                	ELSIF info.ClampA_Setting.PlaceArea = E_FeedInEmptyBox_PlaceArea.SameSizeConveyor THEN
                    	IF Input.bSameSizeCV_BoxNearStorageSensor THEN
                        	SlideClear_1st := FALSE;
                    	ELSE
                        	SlideClear_1st := TRUE;
                    	END_IF
                	END_IF
					IF SlideClear_1st  THEN
                		uiPlaceBothStep := 40;
					END_IF
//				ELSE
//					SlideClear_1st := FALSE;
//				END_IF
				IF Robot._DI1.Error THEN
					uiResumeStep := 81000;	// 補 missing assignment:雷射觸發 Robot.Error 走這條 abort 路徑時,uiResumeStep 必須設成本 step,否則 ABORTING/ABORTED 會用前一階段(pickup)的舊值,resume 跳回 pickup → 撞機
					uiResumePlaceBothStep := 0;
					SlideClear_1st		  := FALSE;
					_Abort	  := TRUE;
					strStatus := CONCAT('FB_FeedInEmptyBoxWithRobot_V3 Step 81000:',Robot.ErrMsg);
				END_IF
            40: //setup for clampB				
			
				CASE Info.ClampB_Setting.PlaceArea OF
					E_FeedInEmptyBox_PlaceArea.DiffSizeConveyor:
						WorkingConveyor REF= DiffSizeCV;
					E_FeedInEmptyBox_PlaceArea.SameSizeConveyor:
						WorkingConveyor REF= SameSizeCV;
				END_CASE
				IF __ISVALIDREF(WorkingConveyor) THEN
					uiPlaceBothStep := 50;
				END_IF
				IF Robot._DI1.Error THEN
					uiResumeStep := 81000;	// 補 missing assignment:雷射觸發 Robot.Error 走這條 abort 路徑時,uiResumeStep 必須設成本 step,否則 ABORTING/ABORTED 會用前一階段(pickup)的舊值,resume 跳回 pickup → 撞機
					uiResumePlaceBothStep := 0;
					SlideClear_1st		  := FALSE;
					_Abort	  := TRUE;
					strStatus := CONCAT('FB_FeedInEmptyBoxWithRobot_V3 Step 81000:',Robot.ErrMsg);
				END_IF

			50://Wait Robot finish clampA
				IF Robot._DI1.Notification THEN
					uiPlaceBothStep:=60;
				END_IF
				IF Robot._DI1.Error THEN
					uiResumeStep := 81000;	// 補 missing assignment:雷射觸發 Robot.Error 走這條 abort 路徑時,uiResumeStep 必須設成本 step,否則 ABORTING/ABORTED 會用前一階段(pickup)的舊值,resume 跳回 pickup → 撞機
					uiResumePlaceBothStep := 0;
					SlideClear_1st		  := FALSE;
					_Abort	  := TRUE;
					strStatus := CONCAT('FB_FeedInEmptyBoxWithRobot_V3 Step 81000:',Robot.ErrMsg);
				END_IF

			60://Move conveyor forward
				bWorkingConveyorMoveForward:=  TRUE;
				IF WorkingConveyor.InForWard THEN
					uiPlaceBothStep:=70;
				END_IF
				
			70://Update sensor
				M_UpdateConveyorSensor(Info.ClampB_Setting.PlaceArea);
				tonPlaceSensorDelay.IN := NOT SelectedSensor AND WorkingConveyor.InForWard ;
				IF 	tonPlaceSensorDelay.Q THEN
					tonPlaceSensorDelay.IN:=FALSE;
					uiPlaceBothStep:=80;
				END_IF
				
			80://Stop conveyor
				WorkingConveyor.M_MotorStop(); 
				bWorkingConveyorMoveForward:= FALSE;
				bWorkingConveyorMoveBackward :=FALSE; 
//				IF WorkingConveyor.InStopped THEN
//					uiPlaceBothStep:=90;
//				END_IF
				uiPlaceBothStep:=90;
			90:		
				WorkingConveyor.M_MotorStop(); 
				bWorkingConveyorMoveForward:= FALSE;
				bWorkingConveyorMoveBackward :=FALSE; 
//				IF	WorkingConveyor.InStopped THEN
               		 IF info.ClampB_Setting.PlaceArea = E_FeedInEmptyBox_PlaceArea.DiffSizeConveyor THEN
                 	   IF Input.bDifferentSizeCV_BoxDetect7_Sensor THEN						
                    	    SlideClear_2nd := FALSE;
                   		 ELSE                        
							SlideClear_2nd := TRUE;							
                   		 END_IF
					
               		 ELSIF info.ClampB_Setting.PlaceArea = E_FeedInEmptyBox_PlaceArea.SameSizeConveyor THEN
                 	   IF Input.bSameSizeCV_BoxNearStorageSensor THEN
                 	       SlideClear_2nd := FALSE;
                 		ELSE
							SlideClear_2nd := TRUE;
							
                  		END_IF
               			 END_IF
//				END_IF
				
				IF SlideClear_2nd THEN
                	uiPlaceBothStep := 99;
					tonPlaceSensorDelay.IN :=FALSE;
				END_IF
				IF Robot._DI1.Error THEN
						uiResumeStep := 81000;	// 補 missing assignment:雷射觸發 Robot.Error 走這條 abort 路徑時,uiResumeStep 必須設成本 step,否則 ABORTING/ABORTED 會用前一階段(pickup)的舊值,resume 跳回 pickup → 撞機
						uiResumePlaceBothStep := 60;
						SlideClear_2nd		  := FALSE;
						_Abort	  := TRUE;
						strStatus := CONCAT('FB_FeedInEmptyBoxWithRobot_V3 Step 81000:',Robot.ErrMsg);
					END_IF

			99:
				IF Robot._DI1.Error THEN
					uiResumeStep := 81000;	// 補 missing assignment:雷射觸發 Robot.Error 走這條 abort 路徑時,uiResumeStep 必須設成本 step,否則 ABORTING/ABORTED 會用前一階段(pickup)的舊值,resume 跳回 pickup → 撞機
					uiResumePlaceBothStep := 60;
					SlideClear_2nd		  := FALSE;
					_Abort	  := TRUE;
					strStatus := CONCAT('FB_FeedInEmptyBoxWithRobot_V3 Step 81000:',Robot.ErrMsg);
				END_IF
        // wait reset
        END_CASE
		bTimeOutIN :=TRUE;	
        IF NOT Robot._DI1.Done THEN
            Robot.M_StartMoveBoxToFeedInConveyor_ClampBoth(ClampA_Address := info.ClampA_Setting.PlaceArea,
                                                           ClampB_Address := info.ClampB_Setting.PlaceArea,
                                                           SlideClear_1st := SlideClear_1st,
                                                           SlideClear_2nd := SlideClear_2nd);
        ELSE
			bTimeOutIN:=FALSE;
            uiExecutingStep := 90000;
        END_IF
			
		IF tonTimeOut.Q THEN
			bTimeOutIN:=FALSE;
			_Abort :=TRUE;	
			uiResumeStep:=81000;		
			strStatus :='FB_FeedInEmptyBoxWithRobot_V3 Step 81000: Place Box timeout';
		END_IF
		IF Robot._DI1.Error THEN
			bTimeOutIN  := FALSE;
			_Abort 		:= TRUE;
			uiResumeStep:= 81000;
			strStatus	:= concat('FB_FeedInEmptyBoxWithRobot_V3 Step 81000:',Robot.ErrMsg);
			//strStatus	:= 'Test ErrMsg';
		END_IF
	
	90000: // Move conveyor forward a bit
		bWorkingConveyorMoveForward:=TRUE;
		IF WorkingConveyor.InForWard THEN
			uiExecutingStep := 91000;
		END_IF
	
	91000:// DELAY
		tonPlaceSensorDelay.PT:=T#0.8S;
		tonPlaceSensorDelay.IN :=TRUE;
		IF tonPlaceSensorDelay.Q THEN
			uiExecutingStep := 92000;
		END_IF
	
	92000:// STOP MOTOR
		tonPlaceSensorDelay.IN :=FALSE;
		bWorkingConveyorMoveForward:=FALSE;
		WorkingConveyor.M_MotorStop();
		IF WorkingConveyor.InStopped THEN
			uiExecutingStep := 99000;
		END_IF
			
				
    99000: // process done
        // Stop FeedIn conveyor
		tonFeedInConveyorDelay.IN :=TRUE;		//Delay FeedInConveyor stop 500MS Edit by Min
		IF tonFeedInConveyorDelay.Q THEN
			DAS_CoreSys.MachineControl.fballocatearea.M_ReleasePulloutAccess(ControlAccess := E_RoundBeltControlAccess.FanucRobot);
			DiffSizeCV.M_MotorStop();
			SameSizeCV.M_MotorStop();
			bWorkingConveyorMoveForward:=FALSE;
			tonFeedInConveyorDelay.IN :=FALSE;
			Status    := 'FB_FeedInEmptyBoxWithRobot_V3 Step 99000: Process completed';
				IF DiffSizeCV.InStopped AND SameSizeCV.InStopped THEN
				 _Executed := TRUE;
				END_IF
		END_IF
END_CASE

// 移植 mirror V4 (commit 326aa68): _Executed 判斷加 NOT Robot.Halt 防止暫停期間誤跳 DONE;
// 新增 ELSIF Pause 進 STATE_Holding,啟動 PackML 暫停流程
IF _Executed AND NOT Robot.Halt THEN
    eState := STATE_DONE;
ELSIF NOT Execute THEN
    eState := STATE_RESETTING;
ELSIF Pause THEN
	bPauseLatched := TRUE;
	uiPauseFromStep := uiExecutingStep;
	_HoldingCompleted := FALSE;
	_HeldCompleted := FALSE;
	_UnholdCompleted := FALSE;
	uiHoldingStep := 0;
	uiHeldStep := 0;
	uiUnholdStep := 0;
	eState := STATE_Holding;
ELSIF Abort OR _Abort THEN
	//FUN_UniqueErrorCodeGenerator(iErrorID := ErrorID,UinqueErrorCode=>_UniqueErrorCode);
	eState := STATE_ABORTING;
ELSIF _Error THEN
	//FUN_UniqueErrorCodeGenerator(iErrorID := ErrorID,UinqueErrorCode=>_UniqueErrorCode);
	eState := STATE_ERROR;
END_IF
END_METHOD

METHOD M_STATE_HELD
VAR_INPUT
END_VAR
Busy := FALSE;
Paused := TRUE;
Status := 'Paused';

IF NOT Execute THEN
	eState := STATE_RESETTING;
ELSIF Abort OR _Abort THEN
	eState := STATE_ABORTING;
ELSIF _Error THEN
	eState := STATE_ERROR;
ELSIF NOT Pause THEN
	_UnholdCompleted := FALSE;
	uiUnholdStep := 0;
	eState := STATE_UnHold;
END_IF
END_METHOD

METHOD M_STATE_HOLDING
VAR_INPUT
END_VAR
Busy := TRUE;
Paused := FALSE;
Status := 'Pause holding';

bTimeOutIN := FALSE;
tonPlaceSensorDelay.IN := FALSE;
tonFeedInConveyorDelay.IN := FALSE;
bWorkingConveyorMoveForward := FALSE;
bWorkingConveyorMoveBackward := FALSE;

CASE uiHoldingStep OF
	0:
		CASE uiExecutingStep OF
			0,10,20,1000,1100:
				uiHoldingStep := 9999;

			61000,71000,81000,90000,91000,92000:
				IF __ISVALIDREF(WorkingConveyor) THEN
					WorkingConveyor.M_MotorStop();
					IF WorkingConveyor.InStopped THEN
						uiHoldingStep := 9999;
					END_IF
				ELSE
					DiffSizeCV.M_MotorStop();
					SameSizeCV.M_MotorStop();
					IF DiffSizeCV.InStopped AND SameSizeCV.InStopped THEN
						uiHoldingStep := 9999;
					END_IF
				END_IF

			99000:
				DAS_CoreSys.MachineControl.fballocatearea.M_ReleasePulloutAccess(
					ControlAccess := E_RoundBeltControlAccess.FanucRobot);
				DiffSizeCV.M_MotorStop();
				SameSizeCV.M_MotorStop();
				IF DiffSizeCV.InStopped AND SameSizeCV.InStopped THEN
					_Executed := TRUE;
					uiHoldingStep := 9999;
				END_IF

		ELSE
			DAS_CoreSys.MachineControl.fballocatearea.M_StopStoragePulloutAction();
			IF Robot.Halt OR Robot._DI1.Done OR NOT Robot._DI12.BzoneInWork THEN
				uiHoldingStep := 9999;
			END_IF
		END_CASE

	9999:
		_HoldingCompleted := TRUE;
END_CASE

IF NOT Execute THEN
	eState := STATE_RESETTING;
ELSIF Abort OR _Abort THEN
	eState := STATE_ABORTING;
ELSIF _Error THEN
	eState := STATE_ERROR;
ELSIF _Executed THEN
	eState := STATE_DONE;
ELSIF _HoldingCompleted THEN
	eState := STATE_Held;
END_IF
END_METHOD

METHOD  M_STATE_RESETTING
VAR_INPUT
END_VAR
IF _Executed THEN Done :=TRUE ; END_IF
CASE uiResettingStep OF
	0:
		//DAS.fbStorageArea.M_InactivePulloutConveyorInternCtrl();
		Robot.M_ResetAllCommand();
		Robot.Bzone_AllowWork:=FALSE;
		DiffSizeCV.M_MotorStop();
		SameSizeCV.M_MotorStop();
		 DAS_CoreSys.MachineControl.fballocatearea.M_ReleasePulloutAccess(ControlAccess := E_RoundBeltControlAccess.FanucRobot);
		 DAS_CoreSys.MachineControl.fballocatearea.M_StopStoragePulloutAction();
		WareHouse.M_ResetFeedInBox();
		WareHouse.M_ResetReloadBox();
		bWorkingConveyorMoveForward  :=FALSE;
		bWorkingConveyorMoveBackward :=FALSE;
		bTimeOutIN:=FALSE;
		Paused := FALSE;
		bPauseLatched := FALSE;
		uiPauseFromStep := 0;
		AClampMoveDone	:= FALSE;
		BClampMoveDone	:= FALSE;
		_AClampDoingWork	:= FALSE;
		_BClampDoingWork	:= FALSE;
		uiResettingStep := 100;
	100:
		_ResetCompleted := TRUE;
END_CASE
IF _ResetCompleted THEN
    eState := STATE_DORMANT;
END_IF
END_METHOD

METHOD M_STATE_UNHOLD
VAR_INPUT
END_VAR
Paused := FALSE;
Status := '';
tonPlaceSensorDelay.IN := FALSE;
tonFeedInConveyorDelay.IN := FALSE;
_UnholdCompleted := TRUE;

IF _UnholdCompleted THEN
	eState := STATE_EXECUTING;
END_IF
END_METHOD

METHOD PRIVATE M_UpdateConveyorSensor : BOOL
VAR_INPUT
	Area : E_FeedInEmptyBox_PlaceArea;
END_VAR
CASE Area OF
	
	E_FeedInEmptyBox_PlaceArea.SameSizeConveyor :
		SelectedSensor := Input.bSameSizeCV_BoxNearStorageSensor ;
	
	E_FeedInEmptyBox_PlaceArea.DiffSizeConveyor:
		SelectedSensor := Input.bDifferentSizeCV_BoxDetect7_Sensor;
END_CASE
END_METHOD

END_FUNCTION_BLOCK

// ---- Library/20_MachineUnits/21_StorageArea/Service_Robot/FB_ReloadRoundBeltBoxWithRobot_V2.TcPOU
FUNCTION_BLOCK FB_ReloadRoundBeltBoxWithRobot_V2 EXTENDS FB_ObjectBase_V2 IMPLEMENTS IBasicElement
VAR_INPUT
    // Below are the components being controlled.
    Robot         : REFERENCE TO FB_FanucRobot_Basic_V2; // Fanuc Robot
    //AllocatedArea : REFERENCE TO FB_AllocatingSpace; // Allocated area , use to control round belt
	RoundBelt	: REFERENCE TO FB_RoundBeltService;
    WareHouse     : REFERENCE TO FB_WareHouse; // Storage area warehouse A and warehouse B conveyor and sensor
    //	A2_Sensor : REFERENCE TO FB_Sensor;
    //	A3_Sensor : REFERENCE TO FB_Sensor;
	Input : ST_InputTable;
    Info : ST_ReloadRoundBeltBox_Info; // Setting the feedin emptybox action's parameter
    Stop : BOOL;
END_VAR
VAR_OUTPUT
	AClampMoveDone	: BOOL;
	BClampMoveDone	: BOOL;
END_VAR
VAR
    strStatus         : STRING;
    tonTimeOut        : TON;
    tonFeedBoxTimeout : TON;
    _UniqueErrorCode  : STRING;
    PreviousStrStatus : STRING;
    PreviousErrorCode : STRING;
    A2_Sensor         : BOOL;
    A3_Sensor         : BOOL;
	//_Abort			  : BOOL;

	// Clamp work
	_AClampDoingWork	: BOOL;
	_BClampDoingWork	: BOOL;

	// ========== Resume 續做機制 ==========
	uiResumeStep	: UDINT := 0;	// 錯誤發生時記錄的步驟，供續做使用
	
	_bRetry			: BOOL;
END_VAR

SUPER^.A10_StateControl();
A00_BasicUnits();
A2_Sensor := Input.bRoundBelt_ChangeZoneA2Detect_Sensor;
A3_Sensor := Input.bRoundBelt_ChangeZoneA3Detect_Sensor;

(*============================================================
Create Date : 2025/11/22
Last Update	: 2026/03/31
Change Log  : 2025/11/24，send flag A clamp done and B clamp done for C# use to SQL // Owner : Gamin
			  2026/03/31，移植泰興鏡射版本，雷射續做，清除手臂錯誤。
============================================================*)

ACTION A00_BasicUnits:
tonTimeOut(PT:=T#60S);
tonFeedBoxTimeout(PT:=T#15s);
END_ACTION

METHOD M_CheckCommand : BOOL
VAR_INPUT
END_VAR
VAR_INST
	CheckBehavior : BOOL; // True :Behavior is correct
END_VAR
VAR
	I: INT;
END_VAR
// Memory clear
CheckBehavior := FALSE;
// Check command is correct
IF info.ClampA_Setting.Behavior = E_ClampWork.Work OR info.ClampB_Setting.Behavior = E_ClampWork.Work THEN
	CheckBehavior := TRUE;
ELSE
	CheckBehavior := FALSE;
END_IF


M_CheckCommand := CheckBehavior;
END_METHOD

METHOD M_CheckUnitsNotBusy : BOOL
VAR_INPUT
END_VAR
M_CheckUnitsNotBusy := true;
END_METHOD

METHOD M_CheckUnitsReady : BOOL
VAR_INPUT
END_VAR
M_CheckUnitsReady := true;
END_METHOD

METHOD M_SelectActionMode : E_ReloadRoundBoxAction
VAR_INPUT
END_VAR
IF info.ClampA_Setting.Behavior <> E_ClampWork.Work AND info.ClampB_Setting.Behavior <> E_ClampWork.Work THEN
	M_SelectActionMode :=E_ReloadRoundBoxAction.Undefined;
ELSIF info.ClampA_Setting.Behavior = E_ClampWork.Work AND info.ClampB_Setting.Behavior <> E_ClampWork.Work THEN
	IF info.ClampA_Setting.PickUpArea = E_ReloadRoundBelt_PickupArea.WareHouseA THEN
		M_SelectActionMode := E_ReloadRoundBoxAction.ClampA_WareHouseA;
	ELSIF info.ClampA_Setting.PickUpArea = E_ReloadRoundBelt_PickupArea.WareHouseB THEN
		M_SelectActionMode := E_ReloadRoundBoxAction.ClampA_WareHouseB;
	END_IF
ELSIF info.ClampA_Setting.Behavior <> E_ClampWork.Work AND info.ClampB_Setting.Behavior = E_ClampWork.Work THEN
	IF info.ClampB_Setting.PickUpArea = E_ReloadRoundBelt_PickupArea.WareHouseA THEN
		M_SelectActionMode := E_ReloadRoundBoxAction.ClampB_WareHouseA;
	ELSIF info.ClampB_Setting.PickUpArea = E_ReloadRoundBelt_PickupArea.WareHouseB THEN
		M_SelectActionMode := E_ReloadRoundBoxAction.ClampB_WareHouseB;
	END_IF
ELSIF info.ClampA_Setting.Behavior = E_ClampWork.Work AND info.ClampB_Setting.Behavior = E_ClampWork.Work THEN
	IF info.ClampA_Setting.PickUpArea = E_ReloadRoundBelt_PickupArea.WareHouseA THEN
		IF info.ClampB_Setting.PickUpArea = E_ReloadRoundBelt_PickupArea.WareHouseA THEN
			M_SelectActionMode := E_ReloadRoundBoxAction.A_WareHouseA_B_WareHouseA;
		ELSIF info.ClampB_Setting.PickUpArea = E_ReloadRoundBelt_PickupArea.WareHouseB THEN
			M_SelectActionMode := E_ReloadRoundBoxAction.A_WareHouseA_B_WareHouseB;
		END_IF
	ELSIF info.ClampA_Setting.PickUpArea = E_ReloadRoundBelt_PickupArea.WareHouseB THEN
		IF info.ClampB_Setting.PickUpArea = E_ReloadRoundBelt_PickupArea.WareHouseA THEN
			M_SelectActionMode := E_ReloadRoundBoxAction.A_WareHouseB_B_WareHouseA;
		ELSIF info.ClampB_Setting.PickUpArea = E_ReloadRoundBelt_PickupArea.WareHouseB THEN
			M_SelectActionMode := E_ReloadRoundBoxAction.A_WareHouseB_B_WareHouseB;
		END_IF
	END_IF
END_IF
END_METHOD

METHOD  M_STATE_ABORTED
VAR_INPUT
END_VAR
IF NOT _bRetry THEN
	Busy    := FALSE;
	Error	:= TRUE;
	Aborted := TRUE;
	_Abort  := TRUE;
	UniqueErrorCode := _UniqueErrorCode;
	Status := strStatus;
	_AbortCompleted := FALSE;
	uiAbortingStep	:= 0;
END_IF

IF Reset THEN
	_bRetry := TRUE;
	Error	:= FALSE;
	Aborted := FALSE;
	_Abort  := FALSE;
END_IF

// ============================================================
// Resume 機制：保持 Execute 並按 Reset 可從錯誤點繼續
// ============================================================
IF NOT Execute THEN
	eState := STATE_RESETTING;
ELSIF Execute AND _bRetry AND NOT Robot._DI1.Error AND NOT Robot.Halt THEN
	// Resume 模式：確認 Robot 不在暫停且無錯誤，從儲存的步驟繼續執行
	Status := '';

	uiExecutingStep := uiResumeStep;
	PreviousStrStatus := strStatus;
	PreviousErrorCode := _UniqueErrorCode;
	
	IF GVL_ADS.MachineState <>E_MachineState.Error THEN
		eSTATE:=STATE_EXECUTING;
	END_IF
END_IF
END_METHOD

METHOD  M_STATE_ABORTING
VAR_INPUT
END_VAR
CASE uiAbortingStep OF
	0:
			_Abort  := FALSE;
			_bRetry := FALSE;
			tonTimeOut.IN 		 := FALSE;
			tonFeedBoxTimeout.IN := FALSE;

			uiAbortingStep := 100;
	
    100:
			IF Robot._DI1.Error THEN
				uiAbortingStep := 200;
			ELSE
				uiAbortingStep := 9999;
			END_IF
	200:		
			 IF DAS_CoreSys.MachineControl.M_RobotResetCmd() THEN
				 uiAbortingStep := 300;
			 END_IF
	300:
			IF DAS_CoreSys.MachineControl.M_RobotStartCmd() THEN
				 uiAbortingStep := 400;
			 END_IF 
	400:
			IF Robot._DI1.Error THEN
		 		uiAbortingStep := 200;
			ELSE
				uiAbortingStep := 9999;
			END_IF
	9999:
			_AbortCompleted := TRUE;
END_CASE


IF _AbortCompleted THEN
    eState := STATE_Aborted;
END_IF
END_METHOD

METHOD  M_STATE_DONE
VAR_INPUT
END_VAR
Busy   := FALSE;
_Error := Error := FALSE;
_Abort := Abort := FALSE;
Done   := TRUE;

IF NOT Execute THEN
    eState := STATE_RESETTING;
END_IF
END_METHOD

METHOD  M_STATE_DORMANT
VAR_INPUT
END_VAR
// Clear FB output
Busy            := FALSE;
Done            := FALSE;
Aborted         := FALSE;
Error           := FALSE;
ErrorID         := 0;
Status          := '';
_ResetCompleted := FALSE;
_Error          := FALSE;
_Executed       := FALSE;
_Abort			:= FALSE;
uiExecutingStep := 0;
uiResettingStep := 0;
uiResumeStep    := 0;	// 清除 Resume 步驟
uiAbortingStep	:= 0;
tonTimeOut.IN := FALSE;
tonFeedBoxTimeout.IN := FALSE;
PreviousStrStatus := '';
PreviousErrorCode := '';
_UniqueErrorCode := '0';
AClampMoveDone := FALSE;
BClampMoveDone := FALSE;
_AClampDoingWork := FALSE;
_BClampDoingWork := FALSE;
_AbortCompleted	 := FALSE;
_bRetry			 := FALSE;

// Wait Execute command
IF Execute AND NOT stop THEN
    eState := STATE_EXECUTING;
END_IF
END_METHOD

METHOD  M_STATE_ERROR
VAR_INPUT
END_VAR
UniqueErrorCode	:= _UniqueErrorCode;
Error			:= TRUE;
status			:= strStatus;
Busy			:= FALSE;

IF NOT Execute THEN
    eState := STATE_RESETTING;
END_IF
END_METHOD

METHOD M_STATE_EXECUTING
VAR_INPUT
END_VAR
VAR_INST
    ActionMode       : E_ReloadRoundBoxAction;
	BoxReady_1st : BOOL;
	BoxReady_2nd : BOOL;
    CarrierReady_1st : BOOL;
    CarrierReady_2nd : BOOL;
    uiPickUpBothStep : UINT;
    uiPlaceBothStep  : UINT;
    ClampA_WareHouseCoordinates : ST_WareHouseCoordinates;
    ClampB_WareHouseCoordinates : ST_WareHouseCoordinates;
	
	//=============== test only====
		_A2Sensor	:BOOL;
		_A3Sensor	:BOOL;
END_VAR
// Set status busy
Busy := TRUE;
IF THIS^.Stop THEN // Pending the timeout when Stop signal occur
	tonTimeout.IN :=FALSE;
END_IF
CASE uiExecutingStep OF
    0:
        // Clear variable
        ActionMode       := E_ReloadRoundBoxAction.Undefined;
        CarrierReady_1st := FALSE;
        CarrierReady_2nd := FALSE;
        uiPickUpBothStep := 0;
        uiPlaceBothStep  := 0;
		BoxReady_1st := 0;
		BoxReady_2nd := 0;
        // Check command
        IF M_CheckCommand() THEN
            uiExecutingStep := 10;
        END_IF
    10:
        // Start process, check units first
        IF M_CheckUnitsReady() THEN
            uiExecutingStep := 20;
        END_IF
    20:
        // CHeck units not busy state
        IF M_CheckUnitsNotBusy() THEN
            uiExecutingStep := 1000;
        END_IF
    1000:
        // Select action mode
        ActionMode      := M_SelectActionMode();
        uiExecutingStep := 1100;
    1100:
		//DAS_CoreSys.MachineControl.fbAllocateArea.M_ActiveRoundBeltInternalCtrl(); //Request round belt 
		DAS_CoreSys.MachineControl.fbAllocateArea.M_GetRoundBeltAccess(ControlAccess := E_RoundBeltControlAccess.FanucRobot);
        CASE ActionMode OF
            E_ReloadRoundBoxAction.ClampA_WareHouseA:
                uiExecutingStep := 10000;
            E_ReloadRoundBoxAction.ClampA_WareHouseB:
                uiExecutingStep := 11000;
            E_ReloadRoundBoxAction.ClampB_WareHouseA:
                uiExecutingStep := 20000;
            E_ReloadRoundBoxAction.ClampB_WareHouseB:
                uiExecutingStep := 21000;
            E_ReloadRoundBoxAction.A_WareHouseA_B_WareHouseA:
                uiExecutingStep := 30000;
            E_ReloadRoundBoxAction.A_WareHouseA_B_WareHouseB:
                uiExecutingStep := 31000;
            E_ReloadRoundBoxAction.A_WareHouseB_B_WareHouseA:
                uiExecutingStep := 32000;
            E_ReloadRoundBoxAction.A_WareHouseB_B_WareHouseB:
                uiExecutingStep := 33000;
        END_CASE
    10000: // Only ClampA pickup box from WarehouseA
        IF NOT Robot._DI1.Done THEN
            // Read ClampA Warehouse coordinate
            ClampA_WareHouseCoordinates := info.ClampA_Setting.WareHouseSetting;
            // Reload Warehouse target position box
            WareHouse.M_StartReloadBox(WareHouseSelect := E_WareHouse.WareHouseA, WarehouseCoordinates := ClampA_WareHouseCoordinates);

            // Check Box reload completed
            IF WareHouse.bReloadBox_Completed THEN
                BoxReady_1st 	 := TRUE;
				_AClampDoingWork := TRUE;
            END_IF

            // Robot Warehouse move
            Robot.M_StartWareHousePickUpBox_ClampA(WareHouseSelect := E_WareHouse.WareHouseA,
                                                   Info            := ClampA_WareHouseCoordinates,
                                                   BoxReady_1st    := BoxReady_1st);

            DAS_CoreSys.MachineControl.fbAllocateArea.M_GetRoundBeltAccess(ControlAccess := E_RoundBeltControlAccess.FanucRobot);
            DAS_CoreSys.MachineControl.fbAllocateArea.M_StartReloadRoundBeltAtion(ReloadStation := info.ClampA_Setting.RoundBeltSetting.Station);
			
			// make sure robot doing AClamp done
			IF _AClampDoingWork AND  NOT Robot._DI1.ClampA_Open THEN
				AClampMoveDone := TRUE;
			END_IF
        ELSE
			tonTimeOut.IN :=FALSE;
            uiExecutingStep := 10080;
        END_IF
		tonTimeOut.IN :=TRUE;
		IF tonTimeOut.Q THEN
			uiResumeStep := 10000;
			_Abort := TRUE;
			tonTimeOut.IN :=FALSE;
			strStatus :='FB_ReloadRoundBeltBoxWithRobot_V2 Step 10000: Pick Box timeout';
		END_IF
    10080:
        Robot.M_ResetAllCommand(); // Clear command and go to place box
		WareHouse.M_ResetReloadBox();
        IF NOT Robot._DI1.Done THEN
            uiExecutingStep := 60000; // only place clampA
        END_IF
    11000: // Only ClampA pickup box from WarehouseB
        IF NOT Robot._DI1.Done THEN
            // Read ClampA Warehouse coordinate
            ClampA_WareHouseCoordinates := info.ClampA_Setting.WareHouseSetting;
            // Reload Warehouse target position box
            WareHouse.M_StartReloadBox(WareHouseSelect := E_WareHouse.WareHouseB, WarehouseCoordinates := ClampA_WareHouseCoordinates);

            // Check Box reload completed
            IF WareHouse.bReloadBox_Completed THEN
                BoxReady_1st 	 := TRUE;
				_AClampDoingWork := TRUE;
            END_IF

            // Robot Warehouse move
            Robot.M_StartWareHousePickUpBox_ClampA(WareHouseSelect := E_WareHouse.WareHouseB,
                                                   Info            := ClampA_WareHouseCoordinates,
                                                   BoxReady_1st    := BoxReady_1st);

            DAS_CoreSys.MachineControl.fbAllocateArea.M_GetRoundBeltAccess(ControlAccess := E_RoundBeltControlAccess.FanucRobot);
            DAS_CoreSys.MachineControl.fbAllocateArea.M_StartReloadRoundBeltAtion(ReloadStation := info.ClampA_Setting.RoundBeltSetting.Station);
			
			// make sure robot doing AClamp done
			IF _AClampDoingWork AND  NOT Robot._DI1.ClampA_Open THEN
				AClampMoveDone := TRUE;
			END_IF

        ELSE
			tonTimeOut.IN :=FALSE;
            uiExecutingStep := 11080;
        END_IF
		tonTimeOut.IN :=TRUE;
		IF tonTimeOut.Q THEN
			uiResumeStep := 11000;
			_Abort := TRUE;
			tonTimeOut.IN :=FALSE;
			strStatus :='FB_ReloadRoundBeltBoxWithRobot_V2 Step 11000: Pick Box timeout';
		END_IF
    11080:
        Robot.M_ResetAllCommand(); // Clear command and go to place box

        IF NOT Robot._DI1.Done THEN
            uiExecutingStep := 60000; // only place clampA
        END_IF
    20000: // Only ClampB pickup from WarehouseA
        IF NOT Robot._DI1.Done THEN
            // Read ClampA Warehouse coordinate
            ClampB_WareHouseCoordinates := info.ClampB_Setting.WareHouseSetting;
            // Reload Warehouse target position box
            WareHouse.M_StartReloadBox(WareHouseSelect := E_WareHouse.WareHouseA, WarehouseCoordinates := ClampB_WareHouseCoordinates);

            // Check Box reload completed
            IF WareHouse.bReloadBox_Completed THEN
                BoxReady_2nd 	 := TRUE;
				_BClampDoingWork := TRUE;
            END_IF

            // Robot Warehouse move
            Robot.M_StartWareHousePickUpBox_ClampB(WareHouseSelect := E_WareHouse.WareHouseA,
                                                   Info            := ClampB_WareHouseCoordinates,
                                                   BoxReady_2nd    := BoxReady_2nd);

          	DAS_CoreSys.MachineControl.fbAllocateArea.M_GetRoundBeltAccess(ControlAccess := E_RoundBeltControlAccess.FanucRobot);
            DAS_CoreSys.MachineControl.fbAllocateArea.M_StartReloadRoundBeltAtion(ReloadStation := info.ClampB_Setting.RoundBeltSetting.Station);
			
			// robot doing BClamp done
			IF _BClampDoingWork AND NOT Robot._DI1.ClampB_Open THEN 
				BClampMoveDone := TRUE;
			END_IF

        ELSE
			tonTimeOut.IN :=FALSE;
            uiExecutingStep := 20080;
        END_IF
			tonTimeOut.IN :=TRUE;
		IF tonTimeOut.Q THEN
			uiResumeStep := 20000;
			_Abort := TRUE;
			tonTimeOut.IN :=FALSE;
			strStatus :='FB_ReloadRoundBeltBoxWithRobot_V2 Step 20000: Pick Box timeout';
		END_IF
    20080:
        WareHouse.M_ResetReloadBox();
        Robot.M_ResetAllCommand();

        IF NOT Robot._DI1.Done THEN
            uiExecutingStep := 70000; // Only ClampB place box
        END_IF
    21000: // Only ClampB pickup from WarehouseB
        IF NOT Robot._DI1.Done THEN
            // Read ClampA Warehouse coordinate
            ClampB_WareHouseCoordinates := info.ClampB_Setting.WareHouseSetting;
            // Reload Warehouse target position box
            WareHouse.M_StartReloadBox(WareHouseSelect := E_WareHouse.WareHouseB, WarehouseCoordinates := ClampB_WareHouseCoordinates);

            // Check Box reload completed
            IF WareHouse.bReloadBox_Completed THEN
                BoxReady_2nd 	 := TRUE;
				_BClampDoingWork := TRUE;
            END_IF

            // Robot Warehouse move
            Robot.M_StartWareHousePickUpBox_ClampB(WareHouseSelect := E_WareHouse.WareHouseB,
                                                   Info            := ClampB_WareHouseCoordinates,
                                                   BoxReady_2nd    := BoxReady_2nd);
            DAS_CoreSys.MachineControl.fbAllocateArea.M_GetRoundBeltAccess(ControlAccess := E_RoundBeltControlAccess.FanucRobot);
            DAS_CoreSys.MachineControl.fbAllocateArea.M_StartReloadRoundBeltAtion(ReloadStation := info.ClampA_Setting.RoundBeltSetting.Station);
			
			// robot doing BClamp done
			IF _BClampDoingWork AND NOT Robot._DI1.ClampB_Open THEN 
				BClampMoveDone := TRUE;
			END_IF

        ELSE
			tonTimeOut.IN :=FALSE;
            uiExecutingStep := 21080;
        END_IF
			tonTimeOut.IN :=TRUE;
		IF tonTimeOut.Q THEN
			uiResumeStep := 21000;
			_Abort := TRUE;
			tonTimeOut.IN :=FALSE;
			strStatus :='FB_ReloadRoundBeltBoxWithRobot_V2 Step 21000: Pick Box timeout';
		END_IF
    21080:
        WareHouse.M_ResetReloadBox();
        Robot.M_ResetAllCommand();

        IF NOT Robot._DI1.Done THEN
            uiExecutingStep := 70000; // Only ClampB place box
        END_IF
    30000: // ClampA and ClampB pickup box from WarehouseA
        ClampA_WareHouseCoordinates := info.ClampA_Setting.WareHouseSetting;
        ClampB_WareHouseCoordinates := info.ClampB_Setting.WareHouseSetting;

        CASE uiPickUpBothStep OF
            0: // ClampA target slide move the box to front side
                WareHouse.M_StartReloadBox(WareHouseSelect      := E_WareHouse.WareHouseA,
                                           WarehouseCoordinates := ClampA_WareHouseCoordinates);

              	DAS_CoreSys.MachineControl.fbAllocateArea.M_GetRoundBeltAccess(ControlAccess := E_RoundBeltControlAccess.FanucRobot);
                DAS_CoreSys.MachineControl.fbAllocateArea.M_StartReloadRoundBeltAtion(ReloadStation := info.ClampA_Setting.RoundBeltSetting.Station);

                IF WareHouse.bReloadBox_Completed THEN
                    BoxReady_1st     := TRUE;
					_AClampDoingWork := TRUE;
                    uiPickUpBothStep := 10;
                END_IF

            10: // wait Robot Allow continue
                IF Robot._DI1.Notification AND
                    NOT
                    WareHouse._stWarehouseList.ASide_Layers[ClampA_WareHouseCoordinates.Layer].stStatus.bSlides[ClampA_WareHouseCoordinates.Slide]
                    THEN
                    WareHouse.M_ResetReloadBox();

                    IF NOT WareHouse.bReloadBox_Completed THEN
                        uiPickUpBothStep := 20;
                    END_IF

                END_IF
            20: // ClampB target slide move the box to front slide
                WareHouse.M_StartReloadBox(WareHouseSelect := E_WareHouse.WareHouseA, WarehouseCoordinates := ClampB_WareHouseCoordinates);

                IF WareHouse.bReloadBox_Completed THEN
                    BoxReady_2nd     := TRUE;
					_BClampDoingWork := TRUE;
                    uiPickUpBothStep := 99;
                END_IF
            99:
        // wait reset
        END_CASE

        Robot.M_StartWareHousePickUpBox_ClampBoth(WareHouseSelect := E_WareHouse.WareHouseA,
                                                  ClampA_Info     := ClampA_WareHouseCoordinates,
                                                  ClampB_Info     := ClampB_WareHouseCoordinates,
                                                  BoxReady_1st    := BoxReady_1st,
                                                  BoxReady_2nd    := BoxReady_2nd);
												  
		// robot doing AClamp done
			IF _AClampDoingWork AND  NOT Robot._DI1.ClampA_Open THEN
				AClampMoveDone := TRUE;
			END_IF

		// robot doing BClamp done
			IF _BClampDoingWork AND NOT Robot._DI1.ClampB_Open THEN 
				BClampMoveDone := TRUE;
			END_IF										  

        IF Robot._DI1.Done THEN
			tonTimeOut.IN :=FALSE;
            uiExecutingStep := 30080;
        END_IF
			tonTimeOut.IN :=TRUE;
		IF tonTimeOut.Q THEN
			uiResumeStep := 30000;
			_Abort := TRUE;
			tonTimeOut.IN :=FALSE;
			strStatus :='FB_ReloadRoundBeltBoxWithRobot_V2 Step 30000: Pick Box timeout';
		END_IF
    30080: // Check robot command is clear
        WareHouse.M_ResetReloadBox();
        Robot.M_ResetAllCommand();

        IF NOT Robot._DI1.Done THEN
            uiExecutingStep := 80000; // go to place step
        END_IF
    31000: // ClampA pickup from Warehouse A, ClampB pickup from Warehouse B
        IF NOT Robot._DI1.Done THEN
            ClampA_WareHouseCoordinates := info.ClampA_Setting.WareHouseSetting;
            WareHouse.M_StartReloadBox(WareHouseSelect := E_WareHouse.WareHouseA, WarehouseCoordinates := ClampA_WareHouseCoordinates);

            IF WareHouse.bReloadBox_Completed THEN
                BoxReady_1st     := TRUE;
				_AClampDoingWork := TRUE;
            END_IF
			DAS_CoreSys.MachineControl.fbAllocateArea.M_ActiveRoundBeltInternalCtrl();
			DAS_CoreSys.MachineControl.fbAllocateArea.M_StartReloadRoundBeltAtion(ReloadStation := info.ClampA_Setting.RoundBeltSetting.Station);
            Robot.M_StartWareHousePickUpBox_ClampA(WareHouseSelect := E_WareHouse.WareHouseA,
                                                   Info            := ClampA_WareHouseCoordinates,
                                                   BoxReady_1st    := BoxReady_1st);
			
			// robot doing AClamp done
			IF _AClampDoingWork AND  NOT Robot._DI1.ClampA_Open THEN
				AClampMoveDone := TRUE;
			END_IF						   
												   
        ELSE
			tonTimeOut.IN :=FALSE;
            uiExecutingStep := 31080;
        END_IF
			tonTimeOut.IN :=TRUE;
		IF tonTimeOut.Q THEN
			uiResumeStep := 31000;
			_Abort := TRUE;
			tonTimeOut.IN :=FALSE;
			strStatus :='FB_ReloadRoundBeltBoxWithRobot_V2 Step 31000: Pick Box timeout';
		END_IF

    31080:
        Robot.M_ResetAllCommand(); // Clear command and go to place box
		WareHouse.M_ResetReloadBox();
        IF NOT Robot._di1.Done THEN
            uiExecutingStep := 31100; // ClampA pickup finished, ClampB pickup start
        END_IF
    31100:
        IF NOT Robot._di1.Done THEN
            ClampB_WareHouseCoordinates := info.ClampB_Setting.WareHouseSetting;
            WareHouse.M_StartReloadBox(WareHouseSelect := E_WareHouse.WareHouseB, WarehouseCoordinates := ClampB_WareHouseCoordinates);

            IF WareHouse.bReloadBox_Completed THEN
                BoxReady_2nd 	 := TRUE;
				_BClampDoingWork := TRUE;
            END_IF

            Robot.M_StartWareHousePickUpBox_ClampB(WareHouseSelect := E_WareHouse.WareHouseB,
                                                   Info            := ClampB_WareHouseCoordinates,
                                                   BoxReady_2nd    := BoxReady_2nd);
												   
			// robot doing BClamp done
			IF _BClampDoingWork AND NOT Robot._DI1.ClampB_Open THEN 
				BClampMoveDone := TRUE;
			END_IF
												   
        ELSE
			tonTimeOut.IN :=FALSE;
            uiExecutingStep := 31180;
        END_IF
				tonTimeOut.IN :=TRUE;
		IF tonTimeOut.Q THEN
			uiResumeStep := 31100;
			_Abort := TRUE;
			tonTimeOut.IN :=FALSE;
			strStatus :='FB_ReloadRoundBeltBoxWithRobot_V2 Step 31100: Pick Box timeout';
		END_IF
    31180:
        Robot.M_ResetAllCommand(); // Clear command and go to place box

        IF NOT Robot._DI1.Done THEN
            uiExecutingStep := 80000; // only place clampA
        END_IF
    32000: // CLampA pickup from Warehouse B, ClampB pickup from Warehouse A
        IF NOT Robot._DI1.Done THEN
            ClampA_WareHouseCoordinates := info.ClampA_Setting.WareHouseSetting;
            WareHouse.M_StartReloadBox(WareHouseSelect := E_WareHouse.WareHouseB, WarehouseCoordinates := ClampA_WareHouseCoordinates);

            IF WareHouse.bReloadBox_Completed THEN
                BoxReady_1st 	 := TRUE;
				_AClampDoingWork := TRUE;
            END_IF
            DAS_CoreSys.MachineControl.fbAllocateArea.M_GetRoundBeltAccess(ControlAccess := E_RoundBeltControlAccess.FanucRobot);
            DAS_CoreSys.MachineControl.fbAllocateArea.M_StartReloadRoundBeltAtion(ReloadStation := info.ClampA_Setting.RoundBeltSetting.Station);
            Robot.M_StartWareHousePickUpBox_ClampA(WareHouseSelect := E_WareHouse.WareHouseB,
                                                   Info            := ClampA_WareHouseCoordinates,
                                                   BoxReady_1st    := BoxReady_1st);
												   
			// robot doing AClamp done
			IF _AClampDoingWork AND  NOT Robot._DI1.ClampA_Open THEN
				AClampMoveDone := TRUE;
			END_IF									   
												   
        ELSE
			tonTimeOut.IN :=FALSE;
            uiExecutingStep := 32080;
        END_IF
				tonTimeOut.IN :=TRUE;
		IF tonTimeOut.Q THEN
			uiResumeStep := 32000;
			_Abort := TRUE;
			tonTimeOut.IN :=FALSE;
			strStatus :='FB_ReloadRoundBeltBoxWithRobot_V2 Step 32000: Pick Box timeout';
		END_IF

    32080:
        Robot.M_ResetAllCommand(); // Clear command and go to place box
		WareHouse.M_ResetReloadBox();
        IF NOT Robot._di1.Done THEN
            uiExecutingStep := 32100; // ClampA pickup finished, ClampB pickup start
        END_IF
    32100:
        IF NOT Robot._di1.Done THEN
            ClampB_WareHouseCoordinates := info.ClampB_Setting.WareHouseSetting;
            WareHouse.M_StartReloadBox(WareHouseSelect := E_WareHouse.WareHouseA, WarehouseCoordinates := ClampB_WareHouseCoordinates);

            IF WareHouse.bReloadBox_Completed THEN
                BoxReady_2nd 	 := TRUE;
				_BClampDoingWork := TRUE;
            END_IF

            Robot.M_StartWareHousePickUpBox_ClampB(WareHouseSelect := E_WareHouse.WareHouseA,
                                                   Info            := ClampB_WareHouseCoordinates,
                                                   BoxReady_2nd    := BoxReady_2nd);
												   
			// robot doing BClamp done
			IF _BClampDoingWork AND NOT Robot._DI1.ClampB_Open THEN 
				BClampMoveDone := TRUE;
			END_IF									   
												   
        ELSE
			tonTimeOut.IN :=FALSE;
            uiExecutingStep := 32180;
        END_IF
				tonTimeOut.IN :=TRUE;
		IF tonTimeOut.Q THEN
			uiResumeStep := 32100;
			_Abort := TRUE;
			tonTimeOut.IN :=FALSE;
			strStatus :='FB_ReloadRoundBeltBoxWithRobot_V2 Step 32100: Pick Box timeout';
		END_IF

    32180:
        Robot.M_ResetAllCommand(); // Clear command and go to place box
		WareHouse.M_ResetReloadBox();
        IF NOT Robot._DI1.Done THEN
            uiExecutingStep := 80000; // only place clampA
        END_IF
    33000: // Both Clamp pickup from WarehouseB
        ClampA_WareHouseCoordinates := info.ClampA_Setting.WareHouseSetting;
        ClampB_WareHouseCoordinates := info.ClampB_Setting.WareHouseSetting;

        CASE uiPickUpBothStep OF
            0: // ClampA target slide move the box to front side
                WareHouse.M_StartReloadBox(WareHouseSelect      := E_WareHouse.WareHouseB,
                                           WarehouseCoordinates := ClampA_WareHouseCoordinates);

                DAS_CoreSys.MachineControl.fbAllocateArea.M_GetRoundBeltAccess(ControlAccess := E_RoundBeltControlAccess.FanucRobot );
                DAS_CoreSys.MachineControl.fbAllocateArea.M_StartReloadRoundBeltAtion(ReloadStation := info.ClampA_Setting.RoundBeltSetting.Station);

                IF WareHouse.bReloadBox_Completed THEN
                    BoxReady_1st     := TRUE;
					_AClampDoingWork := TRUE;
                    uiPickUpBothStep := 10;
                END_IF

            10: // wait Robot Allow continue
                IF Robot._DI1.Notification AND
                    NOT
                    WareHouse._stWarehouseList.BSide_Layers[ClampA_WareHouseCoordinates.Layer].stStatus.bSlides[ClampA_WareHouseCoordinates.Slide]
                    THEN
                    WareHouse.M_ResetReloadBox();

                    IF NOT WareHouse.bReloadBox_Completed THEN
                        uiPickUpBothStep := 20;
                    END_IF

                END_IF
            20: // ClampB target slide move the box to front slide
                WareHouse.M_StartReloadBox(WareHouseSelect := E_WareHouse.WareHouseB, WarehouseCoordinates := ClampB_WareHouseCoordinates);

                IF WareHouse.bReloadBox_Completed THEN
                    BoxReady_2nd     := TRUE;
					_BClampDoingWork := TRUE;
                    uiPickUpBothStep := 99;
                END_IF
            99:
        // wait reset
        END_CASE

        Robot.M_StartWareHousePickUpBox_ClampBoth(WareHouseSelect := E_WareHouse.WareHouseB,
                                                  ClampA_Info     := ClampA_WareHouseCoordinates,
                                                  ClampB_Info     := ClampB_WareHouseCoordinates,
                                                  BoxReady_1st    := BoxReady_1st,
                                                  BoxReady_2nd    := BoxReady_2nd);
												  
		// robot doing AClamp done
			IF _AClampDoingWork AND  NOT Robot._DI1.ClampA_Open THEN
				AClampMoveDone := TRUE;
			END_IF

		// robot doing BClamp done
			IF _BClampDoingWork AND NOT Robot._DI1.ClampB_Open THEN 
				BClampMoveDone := TRUE;
			END_IF										  
												  

        IF Robot._DI1.Done THEN
			tonTimeOut.IN :=FALSE;
            uiExecutingStep := 33080;
        END_IF
		
			tonTimeOut.IN :=TRUE;
		IF tonTimeOut.Q THEN
			uiResumeStep := 33000;
			_Abort := TRUE;
			tonTimeOut.IN :=FALSE;
			strStatus :='FB_ReloadRoundBeltBoxWithRobot_V2 Step 33000: Pick Box timeout';
		END_IF

    33080:
        WareHouse.M_ResetReloadBox();
        Robot.M_ResetAllCommand();

        IF NOT Robot._DI1.Done THEN
            uiExecutingStep := 80000;
        END_IF
    60000: // Only ClampA place box
        WareHouse.M_ResetReloadBox();
        Robot.M_ResetAllCommand();

        // Check Robot RSR1 not working
        IF NOT Robot._di1.Done AND
            NOT (Robot._DI1.AbsMoveA OR
            Robot._DI1.AbsMoveB OR
            Robot._DI1.WarehouseA OR
            Robot._DI1.WarehouseB) THEN
			DAS_CoreSys.MachineControl.fbAllocateArea.M_GetRoundBeltAccess(ControlAccess := E_RoundBeltControlAccess.FanucRobot);
            uiExecutingStep := 61000;
        END_IF
    61000:
        
				DAS_CoreSys.MachineControl.fbAllocateArea.M_GetRoundBeltAccess(ControlAccess := E_RoundBeltControlAccess.FanucRobot);
				DAS_CoreSys.MachineControl.fbAllocateArea.M_StartReloadRoundBeltAtion(ReloadStation := info.ClampA_Setting.RoundBeltSetting.Station);
				IF RoundBelt.xDone  AND arAxisCtrl_gb[AxisNo.RoundBelt].Admin.Axis.Status.NotMoving THEN	
					DAS_CoreSys.MachineControl.fbAllocateArea.M_ResetReloadRoundBeltAction();	
					CarrierReady_1st:=TRUE;			
				 	uiExecutingStep := 61010;
			    END_IF
				IF RoundBelt.xError THEN
					_Error :=TRUE;
					DAS_CoreSys.MachineControl.fbAllocateArea.M_ResetReloadRoundBeltAction();	
					strStatus:='FB_ReloadRoundBeltBoxWithRobot_V2 Step 61000: RoundBelt Error';
				END_IF
	61010:
			
        IF NOT Robot._DI1.Done THEN
            Robot.M_StartMoveBoxToRoundBelt_ClampA(CarrierSelect := info.ClampA_Setting.RoundBeltSetting.ReloadCarrier,
                                                   A2_Sensor     := A2_Sensor,
                                                   A3_Sensor     := A3_Sensor,
                                                   RoundBeltSafe := CarrierReady_1st);
        ELSE
			tonTimeOut.IN :=FALSE;
            uiExecutingStep := 61080;
        END_IF
			tonTimeOut.IN :=TRUE;
		IF tonTimeOut.Q THEN
			uiResumeStep := 61010;
			_Abort := TRUE;
			tonTimeOut.IN :=FALSE;
			strStatus :='FB_ReloadRoundBeltBoxWithRobot_V2 Step 61010: Place Box timeout';
		END_IF
		IF Robot._DI1.Error THEN
			uiResumeStep := 61010;
			_Abort := TRUE;
			strStatus :=CONCAT(STR1 := 'FB_ReloadRoundBeltBoxWithRobot_V2 Step 61010: ',
							   STR2 := Robot.ErrMsg);
		END_IF

    61080:
		DAS_CoreSys.MachineControl.fbAllocateArea.M_ResetReloadRoundBeltAction();
        DAS_CoreSys.MachineControl.fbAllocateArea.M_ReleaseRoundBeltAccess(ControlAccess := E_RoundBeltControlAccess.FanucRobot);
        Robot.M_ResetAllCommand();

        IF NOT Robot._DI1.Done THEN
            uiExecutingStep := 99000; // Go to process end
        END_IF
    70000: // Only ClampB place box
        WareHouse.M_ResetReloadBox();
        Robot.M_ResetAllCommand();

        // Check Robot RSR1 not working
        IF NOT Robot._di1.Done AND
            NOT (Robot._DI1.AbsMoveA OR
            Robot._DI1.AbsMoveB OR
            Robot._DI1.WarehouseA OR
            Robot._DI1.WarehouseB) THEN
            uiExecutingStep := 71000;
        END_IF
    71000:
        // Active RoundBelt INTERNAL control
//               DAS_CoreSys.MachineControl.fbAllocateArea.M_GetRoundBeltAccess(ControlAccess := E_RoundBeltControlAccess.FanucRobot);
//               DAS_CoreSys.MachineControl.fbAllocateArea.M_StartReloadRoundBeltAtion(ReloadStation := info.ClampB_Setting.RoundBeltSetting.Station);
				IF RoundBelt.xDone THEN
					DAS_CoreSys.MachineControl.fbAllocateArea.M_ResetReloadRoundBeltAction();
					//DAS_CoreSys.MachineControl.fbAllocateArea.M_ReleaseRoundBeltAccess(ControlAccess := E_RoundBeltControlAccess.FanucRobot);
					CarrierReady_2nd :=TRUE;
				 	uiExecutingStep := 71010;
			    END_IF
				IF RoundBelt.xError THEN
					_Error :=TRUE;
					DAS_CoreSys.MachineControl.fbAllocateArea.M_ResetReloadRoundBeltAction();
					DAS_CoreSys.MachineControl.fbAllocateArea.M_ReleaseRoundBeltAccess(ControlAccess := E_RoundBeltControlAccess.FanucRobot);
					strStatus:='FB_ReloadRoundBeltBoxWithRobot_V2 Step 71000: RoundBelt Error';
				END_IF
	71010:
			
        IF NOT Robot._DI1.Done THEN
            Robot.M_StartMoveBoxToRoundBelt_ClampB(CarrierSelect := info.ClampB_Setting.RoundBeltSetting.ReloadCarrier,
                                                   A2_Sensor     := A2_Sensor,
                                                   A3_Sensor     := A3_Sensor,
                                                   RoundBeltSafe := CarrierReady_2nd);
        ELSE
			tonTimeOut.IN :=FALSE;
            uiExecutingStep := 71080;
        END_IF
			tonTimeOut.IN :=TRUE;
		IF tonTimeOut.Q THEN
			uiResumeStep := 71010;
			_Abort := TRUE;
			tonTimeOut.IN :=FALSE;
			strStatus :='FB_ReloadRoundBeltBoxWithRobot_V2 Step 71010: Place Box timeout';
		END_IF
		IF Robot._DI1.Error THEN
			uiResumeStep := 71010;
			_Abort := TRUE;
			strStatus :=CONCAT(STR1 := 'FB_ReloadRoundBeltBoxWithRobot_V2 Step 71010: ',
							   STR2 := Robot.ErrMsg);
		END_IF

    71080:
		DAS_CoreSys.MachineControl.fbAllocateArea.M_ResetReloadRoundBeltAction();
        DAS_CoreSys.MachineControl.fbAllocateArea.M_ReleaseRoundBeltAccess(ControlAccess :=E_RoundBeltControlAccess.FanucRobot );       
        Robot.M_ResetAllCommand();

        IF NOT Robot._DI1.Done THEN
            uiExecutingStep := 99000; // Go to process end
        END_IF
    80000:                            // Both Clamp place box
        WareHouse.M_ResetReloadBox(); // Clear Warehouse reload command
        Robot.M_ResetAllCommand();    // Clear Fanuc Robot command
        IF NOT Robot._DI1.Done THEN
            uiExecutingStep := 81000;
        END_IF;
    81000:
        CASE uiPlaceBothStep OF
            0:
				//=============
				_A2Sensor:=FALSE;
				_A3Sensor:=FALSE;
				//==============
                CarrierReady_1st := FALSE;
                CarrierReady_2nd := FALSE;
				DAS_CoreSys.MachineControl.fbAllocateArea.M_GetRoundBeltAccess(ControlAccess := E_RoundBeltControlAccess.FanucRobot);
                uiPlaceBothStep  := 10;
            10:
                // Check move Round Belt done
                IF RoundBelt.xDone THEN
					DAS_CoreSys.MachineControl.fbAllocateArea.M_ResetReloadRoundBeltAction();
					DAS_CoreSys.MachineControl.fbAllocateArea.M_ReleaseRoundBeltAccess(ControlAccess :=E_RoundBeltControlAccess.FanucRobot );       
                    CarrierReady_1st := TRUE;
                    uiPlaceBothStep  := 11;
                END_IF
				IF RoundBelt.xError THEN
					_Error :=TRUE;
					DAS_CoreSys.MachineControl.fbAllocateArea.M_ResetReloadRoundBeltAction();
					DAS_CoreSys.MachineControl.fbAllocateArea.M_ReleaseRoundBeltAccess(ControlAccess :=E_RoundBeltControlAccess.FanucRobot );       
					strStatus:='FB_ReloadRoundBeltBoxWithRobot_V2 Step 81000: RoundBelt Error';
				END_IF
            11:
				//========================Test==================
				IF info.ClampA_Setting.RoundBeltSetting.ReloadCarrier = E_ReloadRoundBelt_PlaceAddress.A2 AND NOT A2_Sensor THEN
					_A2Sensor		:= A2_Sensor;
					uiPlaceBothStep := 15;
				ELSIF info.ClampA_Setting.RoundBeltSetting.ReloadCarrier = E_ReloadRoundBelt_PlaceAddress.A2 AND  A2_Sensor THEN				//edited By Gamin 2026/04/02，放盒位有盒就報警
					_Abort 	  := TRUE;
					strStatus := 'FB_ReloadRoundBeltBoxWithRobot_V2 Step 81000: ClampA place A2 Position has box';
				END_IF
				IF info.ClampA_Setting.RoundBeltSetting.ReloadCarrier = E_ReloadRoundBelt_PlaceAddress.A3 AND NOT A3_Sensor THEN
					_A3Sensor		:= A3_Sensor;
					uiPlaceBothStep := 15;
				ELSIF info.ClampA_Setting.RoundBeltSetting.ReloadCarrier = E_ReloadRoundBelt_PlaceAddress.A3 AND  A3_Sensor THEN
					_Abort	  := TRUE;
					strStatus := 'FB_ReloadRoundBeltBoxWithRobot_V2 Step 81000: ClampA place A3 Position has box'; 
				END_IF
				
			15:
				//======================End_test==================
                IF ((info.ClampA_Setting.RoundBeltSetting.ReloadCarrier = E_ReloadRoundBelt_PlaceAddress.A2) AND A2_Sensor) OR
                    ((info.ClampA_Setting.RoundBeltSetting.ReloadCarrier = E_ReloadRoundBelt_PlaceAddress.A3) AND A3_Sensor)
                    THEN
					DAS_CoreSys.MachineControl.fbAllocateArea.M_GetRoundBeltAccess(ControlAccess := E_RoundBeltControlAccess.FanucRobot);
                    uiPlaceBothStep :=20;// 30;
                END_IF
            20:
                // Wait Notification
                IF robot._DI1.Notification THEN
					//========================Test==================
						IF info.ClampA_Setting.RoundBeltSetting.ReloadCarrier = E_ReloadRoundBelt_PlaceAddress.A2 THEN
							_A2Sensor:=FALSE;
						END_IF
						IF info.ClampA_Setting.RoundBeltSetting.ReloadCarrier = E_ReloadRoundBelt_PlaceAddress.A3 THEN
							_A3Sensor:=FALSE;
						END_IF
				//======================End_test==================
                    DAS_CoreSys.MachineControl.fbAllocateArea.M_ResetReloadRoundBeltAction();

                    IF NOT RoundBelt.xDone THEN
                        uiPlaceBothStep := 30;
                    END_IF
                END_IF
            30: // Move Round belt 2nd time
				DAS_CoreSys.MachineControl.fbAllocateArea.M_GetRoundBeltAccess(ControlAccess := E_RoundBeltControlAccess.FanucRobot);
				DAS_CoreSys.MachineControl.fbAllocateArea.M_StartReloadRoundBeltAtion(ReloadStation := info.ClampB_Setting.RoundBeltSetting.Station);
                uiPlaceBothStep := 40;
            40:
                IF RoundBelt.xDone THEN
					DAS_CoreSys.MachineControl.fbAllocateArea.M_ResetReloadRoundBeltAction();
                    CarrierReady_2nd := TRUE;
                    uiPlaceBothStep  := 80;
                END_IF
				IF RoundBelt.xError THEN
					_Error :=TRUE;
					DAS_CoreSys.MachineControl.fbAllocateArea.M_ResetReloadRoundBeltAction();	
					strStatus:='FB_ReloadRoundBeltBoxWithRobot_V2 Step 81000: RoundBelt Error';
				END_IF
            80:	
				//========================Test==================
				IF info.ClampB_Setting.RoundBeltSetting.ReloadCarrier = E_ReloadRoundBelt_PlaceAddress.A2 AND NOT A2_Sensor THEN
					_A2Sensor:=A2_Sensor;
					uiPlaceBothStep := 99;
				ELSIF info.ClampB_Setting.RoundBeltSetting.ReloadCarrier = E_ReloadRoundBelt_PlaceAddress.A2 AND  A2_Sensor THEN
					_Abort	  := TRUE;
					strStatus := 'FB_ReloadRoundBeltBoxWithRobot_V2 Step 81000: ClampB place A2 Position has box'; 
				END_IF
				IF info.ClampB_Setting.RoundBeltSetting.ReloadCarrier = E_ReloadRoundBelt_PlaceAddress.A3 AND NOT A3_Sensor THEN
					_A3Sensor:=A3_Sensor;
					uiPlaceBothStep := 99;
				ELSIF info.ClampB_Setting.RoundBeltSetting.ReloadCarrier = E_ReloadRoundBelt_PlaceAddress.A3 AND  A3_Sensor THEN
					_Abort	  := TRUE;
					strStatus := 'FB_ReloadRoundBeltBoxWithRobot_V2 Step 81000: ClampB place A3 Position has box'; 
				END_IF
				//======================End_test==================
			99:
				;
			
        // wait reset
        END_CASE

        IF NOT Robot._DI1.Done THEN
            Robot.M_StartMoveBoxToRoundBelt_Both(CarrierSelect_ClampA := info.ClampA_Setting.RoundBeltSetting.ReloadCarrier,
                                                 CarrierSelect_ClampB := info.ClampB_Setting.RoundBeltSetting.ReloadCarrier,
                                                 A2_Sensor            := _A2Sensor,//A2_Sensor,
                                                 A3_Sensor            := _A3Sensor,//A3_Sensor,
                                                 RoundBeltSafe_1st    := CarrierReady_1st,
                                                 RoundBeltSafe_2nd    := CarrierReady_2nd);
        ELSE
			tonTimeOut.IN :=FALSE;
            uiExecutingStep := 99000;
        END_IF
			tonTimeOut.IN :=TRUE;
		IF tonTimeOut.Q THEN
			uiResumeStep := 81000;
			_Abort := TRUE;
			tonTimeOut.IN :=FALSE;
			strStatus :='FB_ReloadRoundBeltBoxWithRobot_V2 Step 81000: Place Box timeout';
		END_IF
		IF Robot._DI1.Error THEN
			uiResumeStep := 81000;
			_Abort		 := TRUE;
			strStatus	 := CONCAT(STR1 := 'FB_ReloadRoundBeltBoxWithRobot_V2 Step 81000: ',
								   STR2 := Robot.ErrMsg);
		END_IF
		
    99000: // process done

			DAS_CoreSys.MachineControl.fbAllocateArea.M_ResetReloadRoundBeltAction();
			DAS_CoreSys.MachineControl.fbAllocateArea.M_ReleaseRoundBeltAccess(ControlAccess :=E_RoundBeltControlAccess.FanucRobot );       
        	Status    := 'FB_ReloadRoundBeltBoxWithRobot_V2 Step 99000: Process completed';
        	_Executed := TRUE;
END_CASE

IF _Executed THEN
    eState := STATE_DONE;
ELSIF NOT Execute THEN
    eState := STATE_RESETTING;
ELSIF Abort OR _Abort THEN
	eState :=STATE_ABORTING;
ELSIF _Error THEN
	eState :=STATE_ERROR;
END_IF
END_METHOD

METHOD  M_STATE_RESETTING
VAR_INPUT
END_VAR
// Done := false 更改到Dormant 清除確保，上位檢查到done 後可以直接下Execute

CASE uiResettingStep OF
	0:
		AClampMoveDone	:= FALSE;
		BClampMoveDone	:= FALSE;
		_AClampDoingWork	:= FALSE;
		_BClampDoingWork	:= FALSE;
		DAS_CoreSys.MachineControl.fbAllocateArea.M_ResetReloadRoundBeltAction();
		DAS_CoreSys.MachineControl.fbAllocateArea.M_ReleaseRoundBeltAccess(ControlAccess :=E_RoundBeltControlAccess.FanucRobot );
		WareHouse.M_ResetReloadBox();
		Robot.M_ResetAllCommand();
		uiResettingStep := 100;
	100:
//		Done := FALSE;
//		Busy := FALSE;
		_ResetCompleted := TRUE;
END_CASE
IF _ResetCompleted THEN
    eState := STATE_DORMANT;
END_IF
END_METHOD

END_FUNCTION_BLOCK

// ---- Library/20_MachineUnits/21_StorageArea/Service_Robot/FB_RobotRegionMove_AllocatedConveyor.TcPOU
FUNCTION_BLOCK FB_RobotRegionMove_AllocatedConveyor EXTENDS FB_ObjectBase_V2 IMPLEMENTS IBasicElement
VAR_INPUT
    Robot     					: REFERENCE TO FB_FanucRobot_Basic_V2;
	DifferenceCV 				: REFERENCE TO FB_motor;    // Allocated area feed in conveyor(diff and same size conveyor)
	SamesizeCV					: REFERENCE TO FB_motor;
//	SameSizeFullSensor 			: REFERENCE TO BOOL; 				 // Because the same size sensor implement FB_ConveyorSameSize, so use reference to connect it
   // Command   : ST_WareHouseWithRobotMove_Command;
   	cylinder : REFERENCE TO UNI_CylinderList;
   	Input : ST_InputTable;
    Info	  : ST_RobotRegionMove_Info;
	Stop	  : BOOL;
END_VAR
VAR_OUTPUT
  // Status : ST_WareHouseWithRobotMove_Status;
END_VAR
VAR
	//_Abort		: BOOL;
	strStatus	: STRING;
	uiResumeStep : UINT;
	
	Area	: E_RobotArea :=E_RobotArea.TransmitCV;
	UseA 	: BOOL;
	UseB	: BOOL;
	SameSizeFullSensor 			: BOOL; 				 // Because the same size sensor implement FB_ConveyorSameSize, so use reference to connect it
	Get 	:BOOL;
	tonTimeOut	:TON;
	tonDelay	:TON;
	tonDelay_SameSizeGetBox 	: TON;
	tonDelay_SameSizeDelayBox 	: TON;
	tonFeedBoxTimeout 			: TON;
	TON_CVmovedelay				: TON;
	_UniqueErrorCode :STRING;
	PreviousStrStatus : STRING;
	PreviousErrorCode : STRING;
	
	_bRetry	: BOOL;
END_VAR

SUPER^.A10_StateControl();
A00_BasicUnits();
SameSizeFullSensor := Input.bSameSizeCV_BoxNearStorageSensor;

(*============================================================
Create Date : 2026/04/01
Last Update	: 2026/04/01
Change Log  : 2026/04/01，移植泰興鏡射機版本。
============================================================*)

ACTION A00_BasicUnits:
tonTimeOut(PT:=T#60S);
tonFeedBoxTimeout(PT:=T#30s);
tonDelay(PT:=T#1.5S);
tonDelay_SameSizeDelayBox(PT:=T#1.5S);
tonDelay_SameSizeGetBox(PT:=T#50MS);
TON_CVmovedelay(PT:= T#1S);
ErrorID:=2210;
END_ACTION

METHOD M_CheckClampStatus : BOOL
VAR_INPUT
END_VAR
M_CheckClampStatus := FALSE;

IF NOT UseA AND NOT UseB THEN
	M_CheckClampStatus 	:= FALSE;
	strStatus 			:= 'FB_RobotRegionMove_AllocatedConveyor: Wrong Command , Both Clammp not used';
	RETURN;
END_IF

IF UseA THEN
	IF Get THEN
		IF NOT Robot._DI1.ClampA_Open THEN
			M_CheckClampStatus  := FALSE;
			strStatus			:= 'FB_RobotRegionMove_AllocatedConveyor: Robot Use A Clamp Get ,but Clamp not open ';
			RETURN;
		END_IF
	ELSE
		IF Robot._DI1.ClampA_Open THEN
			M_CheckClampStatus	:= FALSE;
			strStatus			:= 'FB_RobotRegionMove_AllocatedConveyor: Robot Use A Clamp Place ,but Clamp open';
			RETURN;
		END_IF
	END_IF
END_IF
IF UseB THEN
	IF Get THEN
		IF NOT Robot._DI1.ClampB_Open THEN
			M_CheckClampStatus  := FALSE;
			strStatus			:= 'FB_RobotRegionMove_AllocatedConveyor: Robot Use B Clamp Get ,but Clamp not open ';
			RETURN;
		END_IF
	ELSE
		IF Robot._DI1.ClampB_Open THEN
			M_CheckClampStatus	:= FALSE;
			strStatus			:= 'FB_RobotRegionMove_AllocatedConveyor: Robot Use B Clamp Place ,but Clamp open';
			RETURN;
		END_IF
	END_IF
END_IF

M_CheckClampStatus := TRUE;
END_METHOD

METHOD M_CheckCommand : BOOL // True : Command is useful
VAR_INPUT
END_VAR
VAR
	
END_VAR
// Check command paremeter is correct
	
	THIS^.Get :=Info.Get;	
	UseA :=Info.UseA;
	UseB :=Info.UseB;
	
//Allocated/Empty conveyor
		IF UseA AND ( Info.A_Position<1 OR  Info.A_Position>2 ) THEN
			strStatus:='FB_RobotRegionMove_AllocatedConveyor: Wrong command ,Position A Not allow';
			M_CheckCommand:=FALSE;
			RETURN;		
		END_IF
	
		IF UseB AND ( Info.B_Position<1 OR  Info.B_Position>2 )THEN
			strStatus:='FB_RobotRegionMove_AllocatedConveyor: Wrong command ,Position B Not allow';
			M_CheckCommand:=FALSE;
			RETURN;		
		END_IF	
M_CheckCommand:=TRUE;
END_METHOD

METHOD M_CheckUnitsNotBusy : BOOL
VAR_INPUT
END_VAR
M_CheckUnitsNotBusy := true;
END_METHOD

METHOD M_CheckUnitsReady : BOOL
VAR_INPUT
END_VAR
M_CheckUnitsReady := true;
END_METHOD

METHOD  M_STATE_ABORTED
VAR_INPUT
END_VAR
IF NOT _bRetry THEN
	ERROR 	:= TRUE;
	Busy    := FALSE;
	Aborted := TRUE;
	Status 	:= strStatus;
	UniqueErrorCode:=_UniqueErrorCode;
	_AbortCompleted:= FALSE;
	uiAbortingStep := 0;
END_IF

IF reset THEN
	_bRetry := TRUE;
	ERROR 	:= FALSE;
	Aborted := FALSE;
	_Abort 	:= FALSE;
END_IF


IF NOT Execute THEN
	eSTATE:=STATE_RESETTING;
END_IF

IF Execute AND _bRetry AND NOT Robot._DI1.Error AND NOT Robot.Halt THEN
	status := '';
	uiExecutingStep   := uiResumeStep;
	PreviousStrStatus := strStatus;
	PreviousErrorCode := _UniqueErrorCode;

	IF GVL_ADS.MachineState <>E_MachineState.Error THEN
		eSTATE:=STATE_EXECUTING;
	END_IF
END_IF
END_METHOD

METHOD  M_STATE_ABORTING
VAR_INPUT
END_VAR
CASE uiAbortingStep OF
	0 :
			tonFeedBoxTimeout.IN 	:= FALSE;
			tonTimeOut.IN 			:= FALSE;
			tonDelay.IN 			:= FALSE;
			TON_CVmovedelay.IN 		:= FALSE;
			_Abort := FALSE;
			_bRetry:= FALSE;
			
			DifferenceCV.M_MotorStop();
			SamesizeCV.M_MotorStop();
			IF strStatus = PreviousStrStatus THEN
				_UniqueErrorCode :=PreviousErrorCode;
			END_IF
			uiAbortingStep:=100;
	100:
			IF Robot._DI1.Error THEN
				uiAbortingStep := 200;
			ELSE
				uiAbortingStep := 9999;
			END_IF
	200:		
			 IF DAS_CoreSys.MachineControl.M_RobotResetCmd() THEN
				 uiAbortingStep := 300;
			 END_IF
	300:
			IF DAS_CoreSys.MachineControl.M_RobotStartCmd() THEN
				 uiAbortingStep := 400;
			 END_IF 
	400:
			IF Robot._DI1.Error THEN
		 		uiAbortingStep := 200;
			ELSE
				uiAbortingStep := 9999;
			END_IF
	9999:	_AbortCompleted:=TRUE;
END_CASE

IF NOT Execute THEN
	eState := STATE_RESETTING;
ELSIF _AbortCompleted THEN
	eState := STATE_Aborted;
END_IF
END_METHOD

METHOD  M_STATE_DONE
VAR_INPUT
END_VAR
Busy   := FALSE;
_Error := Error := FALSE;
_Abort := Abort := FALSE;
Done   := TRUE;

IF NOT Execute THEN
    eState := STATE_RESETTING;
END_IF
END_METHOD

METHOD  M_STATE_DORMANT
VAR_INPUT
END_VAR
// Clear FB output
Busy            := FALSE;
Done            := FALSE;
Aborted         := FALSE;
Error           := FALSE;
ErrorID         := 0;
Status          := '';
_ResetCompleted := FALSE;
_Error          := FALSE;
_Executed       := FALSE;
_Abort			:= FALSE;
tonDelay_SameSizeGetBox.IN := FALSE;
tonDelay_SameSizeDelayBox.IN :=false;
tonTimeOut.IN:=FALSE;
strStatus :='No Error';
uiExecutingStep :=uiResettingStep :=uiResumeStep :=0;
tonDelay.IN :=FALSE;
tonFeedBoxTimeout.IN :=FALSE;
TON_CVmovedelay.IN := FALSE;
_UniqueErrorCode :='0';
PreviousStrStatus			 :='';
PreviousErrorCode			 :='';
_AbortCompleted := FALSE;
_Abort := FALSE;
uiAbortingStep := 0;
_bRetry := FALSE;
// Wait Execute command
IF Execute AND NOT stop THEN
    eState := STATE_EXECUTING;
END_IF
END_METHOD

METHOD  M_STATE_ERROR
VAR_INPUT
END_VAR
ERROR   :=TRUE;
Busy	:=FALSE;
Status := strStatus;
UniqueErrorCode:=_UniqueErrorCode;
DifferenceCV.M_MotorStop();
SamesizeCV.M_MotorStop();
cylinder.List.fbSameSizeCV_Press3.M_Retract();
cylinder.List.fbSameSizeCV_Press4.M_Retract();
IF NOT Execute THEN	
eSTATE:=STATE_RESETTING;
END_IF
END_METHOD

METHOD  M_STATE_EXECUTING
VAR_INPUT
END_VAR
VAR_INST
	BoxReady_1st : BOOL;
	BoxReady_2nd : BOOL;
    uiBothStep : UINT;
    uiSingleClampStep : UINT;	
	Address_A : INT;
	Address_B : INT;
	bGetBoxInSameSizeConveyor : BOOL;
	uiSameGetBoxStep : UINT;
	bSameSizeCVMoveForward  : BOOL;
	bSameSizeCVMoveBackward : BOOL;
	bDiffCVMoveForward		:BOOL;
	bDiffCVMoveBackward		:BOOL;


END_VAR
VAR
	WareHouse: INT;
	
END_VAR
// Set Busy active edit by johnson
Busy := TRUE;
IF THIS^.Stop THEN // Pending the timeout when Stop signal occur
	tonTimeout.IN :=FALSE;
END_IF

IF bSameSizeCVMoveForward THEN
	IF NOT SamesizeCV.InBackWard THEN
		SamesizeCV.M_MoveForward();
	END_IF
END_IF
IF bSameSizeCVMoveBackward THEN
	IF NOT SamesizeCV.InForWard THEN
	 SamesizeCV.M_MoveBackward();
	END_IF
END_IF
IF bDiffCVMoveForward THEN
	IF NOT DifferenceCV.InBackWard THEN
		DifferenceCV.M_MoveForward();
	END_IF
END_IF
IF bDiffCVMoveBackward THEN
	IF NOT DifferenceCV.InForWard THEN
		DifferenceCV.M_MoveBackward();
	END_IF
END_IF


// Service Process
CASE uiExecutingStep OF
	0:
        // Clear variable
        uiBothStep := 0;
		uiSingleClampStep :=0;
		BoxReady_1st := 0;
		BoxReady_2nd := 0;
		tonTimeOut.IN:=FALSE;
		bSameSizeCVMoveForward  :=FALSE;
		bSameSizeCVMoveBackward :=FALSE;
		bDiffCVMoveForward		:=FALSE;
		bDiffCVMoveBackward		:=FALSE;
        // Check command
        IF M_CheckCommand() THEN
            uiExecutingStep := 10;
		ELSE
			_Error:=TRUE;
        END_IF
    10:
        // Start process, check units first
        IF M_CheckUnitsReady() THEN
            uiExecutingStep := 20;
        END_IF
    20:
        // CHeck units not busy state
        IF M_CheckUnitsNotBusy() THEN
            uiExecutingStep := 30;
        END_IF
		
	30:	// 檢查夾爪狀態。
		IF M_CheckClampStatus() THEN
            uiExecutingStep := 1000;
		ELSE
			_Abort	:= TRUE;
        END_IF
   
	1000:   
			// Read   coordinate
			 Area := THIS^.Area;
 			 Address_A := LREAL_TO_INT(Info.A_Position);
			 Address_B := LREAL_TO_INT(Info.B_Position);
			 bGetBoxInSameSizeConveyor := Get AND ((UseA AND Address_A=2) OR (UseB AND Address_B=2));
			 IF bGetBoxInSameSizeConveyor THEN
				 cylinder.List.fbSameSizeCV_Press3.M_Retract();
				 cylinder.List.fbSameSizeCV_Press4.M_Retract();
			 END_IF
			 uiSameGetBoxStep :=0;
			 tonDelay_SameSizeGetBox.IN:=FALSE;
			IF UseA AND NOT UseB THEN
				//Only clampA
				uiExecutingStep := 10000;
			ELSIF NOT UseA AND UseB THEN
				//Only ClampB 
				uiExecutingStep := 20000;
			ELSIF UseA AND UseB THEN
				//Both Clamps
				uiExecutingStep := 30000;		
			END_IF
       
    10000: // Only ClampA 
        IF NOT Robot._DI1.Done THEN
            
            
			CASE uiSingleClampStep OF
				
				0://
					 IF Get THEN // Get box job
						CASE Address_A OF
							1:
								tonDelay.IN :=Input.bDifferentSizeCV_BoxDetect7_Sensor;
								bDiffCVMoveBackward:=TRUE;
								bDiffCVMoveForward:=FALSE;
								DifferenceCV.M_MoveBackward();
								
							2:
								CASE uiSameGetBoxStep OF
									0:
									//tonDelay.IN :=SameSizeFullSensor;	
									bSameSizeCVMoveBackward := TRUE;
									bSameSizeCVMoveForward := FALSE;
									SamesizeCV.M_MoveBackward();
									cylinder.List.fbSameSizeCV_Press3.M_Retract();
									cylinder.List.fbSameSizeCV_Press4.M_Retract();
									uiSameGetBoxStep :=100;
									
									100:
										tonDelay_SameSizeGetBox.IN := Input.bSameSizeCV_BoxDetect6_Sensor;
										IF tonDelay_SameSizeGetBox.Q THEN
											cylinder.List.fbSameSizeCV_Press3.M_Extend();
											uiSameGetBoxStep :=200;
										END_IF
									200:
										tonDelay_SameSizeGetBox.IN:=FALSE;
										tonDelay_SameSizeDelayBox.IN :=SameSizeFullSensor;
										IF 	tonDelay_SameSizeDelayBox.Q THEN
												uiSameGetBoxStep :=300;
										END_IF	
									300:
										cylinder.List.fbSameSizeCV_Press4.M_Extend();
										IF NOT Input.bSameSizeCV_BoxDetect6_Sensor THEN
											tonDelay.IN :=TRUE;
											uiSameGetBoxStep := 400;
										ELSE
											cylinder.List.fbSameSizeCV_Press3.M_Retract();
											bSameSizeCVMoveBackward := FALSE;
											bSameSizeCVMoveForward 	:= FALSE;
											SamesizeCV.M_MotorStop();
											uiSameGetBoxStep := 325;
										END_IF
									325:
										bSameSizeCVMoveBackward := FALSE;
										bSameSizeCVMoveForward 	:= TRUE;
										IF SamesizeCV.InForWard THEN
											uiSameGetBoxStep := 350;
										END_IF
										
									350:
										TON_CVmovedelay.IN := NOT Input.bSameSizeCV_BoxDetect6_Sensor;
										IF TON_CVmovedelay.Q THEN
											cylinder.List.fbSameSizeCV_Press3.M_Extend();
											bSameSizeCVMoveBackward := FALSE;
											bSameSizeCVMoveForward 	:= FALSE;
											SamesizeCV.M_MotorStop();
											uiSameGetBoxStep := 375;
										END_IF
									375:
										TON_CVmovedelay.IN 		:= FALSE;
										bSameSizeCVMoveBackward := TRUE;
										bSameSizeCVMoveForward  := FALSE;
										IF SamesizeCV.InBackWard THEN
											uiSameGetBoxStep := 400;
										END_IF
									400: 
										tonDelay.IN :=TRUE;
										IF tonDelay.Q THEN
											cylinder.List.fbSameSizeCV_Press4.M_Retract();
										END_IF
								END_CASE
						END_CASE	
			
					ELSE
						CASE Address_A OF
							1:
								tonDelay.IN := NOT Input.bDifferentSizeCV_BoxDetect7_Sensor;
								bDiffCVMoveForward :=TRUE;
								bDiffCVMoveBackward:=FALSE;
								DifferenceCV.M_MoveForward();
							2:
								tonDelay.IN :=NOT SameSizeFullSensor;
								bSameSizeCVMoveForward :=TRUE;
								bSameSizeCVMoveBackward:=FALSE;
								SamesizeCV.M_MoveForward();			
						END_CASE					
				
					END_IF	
				
						IF tonDelay.Q THEN
							tonFeedBoxTimeout.IN :=FALSE;
							uiSingleClampStep:=1000;
						END_IF
						tonFeedBoxTimeout.IN :=TRUE;
						IF tonFeedBoxTimeout.Q THEN
							tonFeedBoxTimeout.IN :=FALSE;
							strStatus :='FB_RobotRegionMove_AllocatedConveyor Step 10000: Feed Box timeout';
							uiResumeStep:=10000;
							_Abort:=TRUE;
						END_IF
				1000:
						BoxReady_1st:=TRUE;
						tonDelay.IN:=FALSE;
						bSameSizeCVMoveForward  :=FALSE;
						bSameSizeCVMoveBackward :=FALSE;
						bDiffCVMoveForward		:=FALSE;
						bDiffCVMoveBackward		:=FALSE;						
						DifferenceCV.M_MotorStop();
						SamesizeCV.M_MotorStop();
						uiSingleClampStep:=9999;
				9999: //Wait	
			END_CASE
			          		 
				  // Robot Abs move
           		 Robot.M_StartRobotAbsMove(GetBox:=Get,
											UseClampA:=UseA,
											UseClampB:=UseB,
											Area:=Area,
											ClampA_Address:=Address_A,
											ClampB_Address:=Address_B,
											BoxReady_1:=BoxReady_1st,
											BoxReady_2:=BoxReady_2nd);				  
		
        ELSE
			tonTimeOut.IN:=FALSE;
            uiExecutingStep := 10080;
        END_IF
		tonTimeOut.IN:=TRUE;
		IF tonTimeOut.Q=TRUE THEN
			tonTimeOut.IN:=FALSE;
			strStatus := 'FB_RobotRegionMove_AllocatedConveyor Step 10000: Robot move timeout';
			uiResumeStep := 10000;
			_Abort :=TRUE;
		END_IF	
		IF Robot._DI1.Error THEN
			_Abort	  	 := TRUE;
			strStatus 	 := CONCAT('FB_RobotRegionMove_AllocatedConveyor Step 10000: ',Robot.ErrMsg);
			uiResumeStep := 10000;
		END_IF	
    10080:
        Robot.M_ResetRobotAbsMove(UseA,UseB); // Clear command and go to place box
		tonTimeOut.IN:=TRUE;
		uiSameGetBoxStep:=0;
        IF NOT Robot._DI1.Done THEN
			tonTimeOut.IN:=FALSE;
            uiExecutingStep := 50000; 
        END_IF
		
    	IF tonTimeOut.Q=TRUE THEN
			strStatus :='FB_RobotRegionMove_AllocatedConveyor Step 10080: Reset Robot timeout';
			_Error:=TRUE;
		END_IF	
    
   20000: // Only ClampB
        IF NOT Robot._DI1.Done THEN
            			
			CASE uiSingleClampStep OF
			0:	
					 IF Get THEN // Get box job
						CASE Address_B OF
							1:
								tonDelay.IN :=Input.bDifferentSizeCV_BoxDetect7_Sensor;
								bDiffCVMoveBackward:=TRUE;
								bDiffCVMoveForward := FALSE;
								DifferenceCV.M_MoveBackward();
								
							2:
								CASE uiSameGetBoxStep OF
									0:
									bSameSizeCVMoveForward :=FALSE;
									bSameSizeCVMoveBackward := TRUE;
									SamesizeCV.M_MoveBackward();
									cylinder.List.fbSameSizeCV_Press3.M_Retract();
									cylinder.List.fbSameSizeCV_Press4.M_Retract();
									uiSameGetBoxStep :=100;
									
									100:
										tonDelay_SameSizeGetBox.IN := Input.bSameSizeCV_BoxDetect6_Sensor;
										IF tonDelay_SameSizeGetBox.Q THEN
											cylinder.List.fbSameSizeCV_Press3.M_Extend();
											uiSameGetBoxStep :=200;
										END_IF
									200:
										tonDelay_SameSizeGetBox.IN:=FALSE;
										tonDelay_SameSizeDelayBox.IN :=SameSizeFullSensor;
										IF 	tonDelay_SameSizeDelayBox.Q THEN
											uiSameGetBoxStep :=300;
										END_IF	
									300:
										cylinder.List.fbSameSizeCV_Press4.M_Extend();
										IF NOT Input.bSameSizeCV_BoxDetect6_Sensor THEN
											tonDelay.IN :=TRUE;
											uiSameGetBoxStep := 400;
										ELSE
											cylinder.List.fbSameSizeCV_Press3.M_Retract();
											bSameSizeCVMoveBackward := FALSE;
											bSameSizeCVMoveForward 	:= FALSE;
											SamesizeCV.M_MotorStop();
											uiSameGetBoxStep := 325;
										END_IF
									325:
										bSameSizeCVMoveBackward := FALSE;
										bSameSizeCVMoveForward 	:= TRUE;
										IF SamesizeCV.InForWard THEN
											uiSameGetBoxStep := 350;
										END_IF
										
									350:
										TON_CVmovedelay.IN := NOT Input.bSameSizeCV_BoxDetect6_Sensor;
										IF TON_CVmovedelay.Q THEN
											cylinder.List.fbSameSizeCV_Press3.M_Extend();
											bSameSizeCVMoveBackward := FALSE;
											bSameSizeCVMoveForward 	:= FALSE;
											SamesizeCV.M_MotorStop();
											uiSameGetBoxStep := 375;
										END_IF
									375:
										TON_CVmovedelay.IN 		:= FALSE;
										bSameSizeCVMoveBackward := TRUE;
										bSameSizeCVMoveForward  := FALSE;
										IF SamesizeCV.InBackWard THEN
											uiSameGetBoxStep := 400;
										END_IF
									400: 
										tonDelay.IN :=TRUE;
										IF tonDelay.Q THEN
											cylinder.List.fbSameSizeCV_Press4.M_Retract();
										END_IF
								END_CASE			

						END_CASE	
			
					ELSE
						CASE Address_B OF
							1:
								tonDelay.IN := NOT Input.bDifferentSizeCV_BoxDetect7_Sensor;
								bDiffCVMoveForward	:=TRUE;
								bDiffCVMoveBackward	:=FALSE;
								DifferenceCV.M_MoveForward();
							2:
								tonDelay.IN :=NOT SameSizeFullSensor;
								bSameSizeCVMoveForward :=TRUE;
								bSameSizeCVMoveBackward :=FALSE;
								SamesizeCV.M_MoveForward();			
						END_CASE					
				
					END_IF	
				
						IF tonDelay.Q THEN
							tonFeedBoxTimeout.IN :=FALSE;
							uiSingleClampStep:=1000;
						END_IF
						tonFeedBoxTimeout.IN :=TRUE;
						IF tonFeedBoxTimeout.Q THEN
							tonFeedBoxTimeout.IN :=FALSE;
							strStatus :='FB_RobotRegionMove_AllocatedConveyor Step 20000: Feed Box timeout';
							uiResumeStep:=20000;
							_Abort:=TRUE;
						END_IF
				1000:
						//BoxReady_1st:=TRUE;
						BoxReady_2nd:=TRUE;
						tonDelay.IN:=FALSE;
						bSameSizeCVMoveForward  :=FALSE;
						bSameSizeCVMoveBackward :=FALSE;
						bDiffCVMoveForward		:=FALSE;
						bDiffCVMoveBackward		:=FALSE;
						DifferenceCV.M_MotorStop();
						SamesizeCV.M_MotorStop();
						uiSingleClampStep:=9999;
				9999: //Wait	

			END_CASE
			          		 
				  // Robot Abs move
           		 Robot.M_StartRobotAbsMove( GetBox:=Get,
											UseClampA:=UseA,
											UseClampB:=UseB,
											Area:=Area,
											ClampA_Address:=Address_A,
											ClampB_Address:=Address_B,
											BoxReady_1:=BoxReady_1st,
											BoxReady_2:=BoxReady_2nd);	
        ELSE
			tonTimeOut.IN:=FALSE;
            uiExecutingStep := 20080;
        END_IF
		tonTimeOut.IN:=TRUE;
		IF tonTimeOut.Q=TRUE THEN
			tonTimeOut.IN:=FALSE;
			strStatus := 'FB_RobotRegionMove_AllocatedConveyor Step 20000: Robot move timeout';
			uiResumeStep := 20000;
			_Abort :=TRUE;
		END_IF	
		IF Robot._DI1.Error THEN
			_Abort	  	 := TRUE;
			strStatus 	 := CONCAT('FB_RobotRegionMove_AllocatedConveyor Step 20000: ',Robot.ErrMsg);
			uiResumeStep := 20000;
		END_IF	
    20080:
       Robot.M_ResetRobotAbsMove(UseA,UseB);; // Clear command 
		uiSameGetBoxStep :=0;
        IF NOT Robot._DI1.Done THEN
            uiExecutingStep := 50000; 
        END_IF
		tonTimeOut.IN:=TRUE;
		IF tonTimeOut.Q=TRUE THEN
			strStatus :='FB_RobotRegionMove_AllocatedConveyor Step 20080: Reset Robot timeout';
			_Error:=TRUE;
		END_IF	
    30000: // Both Clamps
        		
		
		  CASE uiBothStep OF
           		0://	
					BoxReady_1st := FALSE;
					BoxReady_2nd := FALSE;					
					uiBothStep:=1000;						
				
				1000:
						IF Get THEN // Get box job
							CASE Address_A OF
								1:
									tonDelay.IN :=Input.bDifferentSizeCV_BoxDetect7_Sensor;
									bDiffCVMoveForward	:=FALSE;
									bDiffCVMoveBackward	:=TRUE;
									DifferenceCV.M_MoveBackward();
									
								2:
								CASE uiSameGetBoxStep OF
									0:
									bSameSizeCVMoveForward  :=FALSE;
									bSameSizeCVMoveBackward :=TRUE;
									SamesizeCV.M_MoveBackward();
									cylinder.List.fbSameSizeCV_Press3.M_Retract();
									cylinder.List.fbSameSizeCV_Press4.M_Retract();
									uiSameGetBoxStep :=100;
									
									100:
										tonDelay_SameSizeGetBox.IN := Input.bSameSizeCV_BoxDetect6_Sensor;
										IF tonDelay_SameSizeGetBox.Q THEN
											cylinder.List.fbSameSizeCV_Press3.M_Extend();
											uiSameGetBoxStep :=200;
										END_IF
									200:
										tonDelay_SameSizeGetBox.IN:=FALSE;
										tonDelay_SameSizeDelayBox.IN :=SameSizeFullSensor;
										IF 	tonDelay_SameSizeDelayBox.Q THEN
											uiSameGetBoxStep :=300;
										END_IF	
									300:
										cylinder.List.fbSameSizeCV_Press4.M_Extend();
										IF NOT Input.bSameSizeCV_BoxDetect6_Sensor THEN
											tonDelay.IN :=TRUE;
											uiSameGetBoxStep := 400;
										ELSE
											cylinder.List.fbSameSizeCV_Press3.M_Retract();
											bSameSizeCVMoveBackward := FALSE;
											bSameSizeCVMoveForward 	:= FALSE;
											SamesizeCV.M_MotorStop();
											uiSameGetBoxStep := 325;
										END_IF
									325:
										bSameSizeCVMoveBackward := FALSE;
										bSameSizeCVMoveForward 	:= TRUE;
										IF SamesizeCV.InForWard THEN
											uiSameGetBoxStep := 350;
										END_IF
										
									350:
										TON_CVmovedelay.IN := NOT Input.bSameSizeCV_BoxDetect6_Sensor;
										IF TON_CVmovedelay.Q THEN
											cylinder.List.fbSameSizeCV_Press3.M_Extend();
											bSameSizeCVMoveBackward := FALSE;
											bSameSizeCVMoveForward 	:= FALSE;
											SamesizeCV.M_MotorStop();
											uiSameGetBoxStep := 375;
										END_IF
									375:
										TON_CVmovedelay.IN 		:= FALSE;
										bSameSizeCVMoveBackward := TRUE;
										bSameSizeCVMoveForward  := FALSE;
										IF SamesizeCV.InBackWard THEN
											uiSameGetBoxStep := 400;
										END_IF
									400: 
										tonDelay.IN :=TRUE;
										IF tonDelay.Q THEN
											cylinder.List.fbSameSizeCV_Press4.M_Retract();
										END_IF
								END_CASE
				
							END_CASE	
			
						ELSE
							CASE Address_A OF
								1:
									tonDelay.IN := NOT Input.bDifferentSizeCV_BoxDetect7_Sensor;
									bDiffCVMoveForward	:=TRUE;
									bDiffCVMoveBackward	:=FALSE;
									DifferenceCV.M_MoveForward();
								2:
									tonDelay.IN :=NOT SameSizeFullSensor;
									bSameSizeCVMoveForward  :=TRUE;
									bSameSizeCVMoveBackward :=FALSE;
									SamesizeCV.M_MoveForward();			
							END_CASE					
				
						END_IF	
				
						IF tonDelay.Q THEN
							tonFeedBoxTimeout.IN :=FALSE;
							uiSameGetBoxStep:=0;
							uiBothStep:=2000;
						END_IF
						tonFeedBoxTimeout.IN :=TRUE;
						IF tonFeedBoxTimeout.Q THEN
							tonFeedBoxTimeout.IN :=FALSE;
							strStatus :='FB_RobotRegionMove_AllocatedConveyor Step 30000: Feed Box timeout';
							uiResumeStep:=30000;
							_Abort:=TRUE;
						END_IF
				2000:
						tonDelay.IN :=FALSE;
						bSameSizeCVMoveForward  :=FALSE;
						bSameSizeCVMoveBackward :=FALSE;
						bDiffCVMoveForward		:=FALSE;
						bDiffCVMoveBackward		:=FALSE;
						DifferenceCV.M_MotorStop();
						SamesizeCV.M_MotorStop();
						BoxReady_1st:=TRUE;
						tonDelay_SameSizeGetBox.IN := FALSE;
						tonDelay_SameSizeDelayBox.IN :=FALSE;
						IF Robot._DI1.Notification THEN
							uiBothStep:=3000;
						END_IF
				3000:
						IF Get THEN // Get box job
							CASE Address_B OF
								1:
									tonDelay.IN :=Input.bDifferentSizeCV_BoxDetect7_Sensor;
									bDiffCVMoveForward	:=FALSE;
									bDiffCVMoveBackward :=TRUE;
									DifferenceCV.M_MoveBackward();
									
								2:
									CASE uiSameGetBoxStep OF
									0:
									bSameSizeCVMoveForward :=FALSE;
									bSameSizeCVMoveBackward :=TRUE;
									SamesizeCV.M_MoveBackward();
									cylinder.List.fbSameSizeCV_Press3.M_Retract();
									cylinder.List.fbSameSizeCV_Press4.M_Retract();
									uiSameGetBoxStep :=100;
									
									100:
										tonDelay_SameSizeGetBox.IN := Input.bSameSizeCV_BoxDetect6_Sensor;
										IF tonDelay_SameSizeGetBox.Q THEN
											cylinder.List.fbSameSizeCV_Press3.M_Extend();
											uiSameGetBoxStep :=200;
										END_IF
									200:
										tonDelay_SameSizeGetBox.IN:=FALSE;
										tonDelay_SameSizeDelayBox.IN :=SameSizeFullSensor;
										IF 	tonDelay_SameSizeDelayBox.Q THEN
											uiSameGetBoxStep :=300;
										END_IF	
									300:
										cylinder.List.fbSameSizeCV_Press4.M_Extend();
										IF NOT Input.bSameSizeCV_BoxDetect6_Sensor THEN
											tonDelay.IN :=TRUE;
											uiSameGetBoxStep := 400;
										ELSE
											cylinder.List.fbSameSizeCV_Press3.M_Retract();
											bSameSizeCVMoveBackward := FALSE;
											bSameSizeCVMoveForward 	:= FALSE;
											SamesizeCV.M_MotorStop();
											uiSameGetBoxStep := 325;
										END_IF
									325:
										bSameSizeCVMoveBackward := FALSE;
										bSameSizeCVMoveForward 	:= TRUE;
										IF SamesizeCV.InForWard THEN
											uiSameGetBoxStep := 350;
										END_IF
										
									350:
										TON_CVmovedelay.IN := NOT Input.bSameSizeCV_BoxDetect6_Sensor;
										IF TON_CVmovedelay.Q THEN
											cylinder.List.fbSameSizeCV_Press3.M_Extend();
											bSameSizeCVMoveBackward := FALSE;
											bSameSizeCVMoveForward 	:= FALSE;
											SamesizeCV.M_MotorStop();
											uiSameGetBoxStep := 375;
										END_IF
									375:
										TON_CVmovedelay.IN 		:= FALSE;
										bSameSizeCVMoveBackward := TRUE;
										bSameSizeCVMoveForward  := FALSE;
										IF SamesizeCV.InBackWard THEN
											uiSameGetBoxStep := 400;
										END_IF
									400: 
										tonDelay.IN := TRUE;
										IF tonDelay.Q THEN
											cylinder.List.fbSameSizeCV_Press4.M_Retract();
										END_IF
								END_CASE
							END_CASE	
			
						ELSE
							CASE Address_B OF
								1:
									tonDelay.IN := NOT Input.bDifferentSizeCV_BoxDetect7_Sensor;
									bDiffCVMoveForward	:=TRUE;
									bDiffCVMoveBackward := FALSE;
									DifferenceCV.M_MoveForward();
								2:
									tonDelay.IN :=NOT SameSizeFullSensor;
									bSameSizeCVMoveForward :=TRUE;
									bSameSizeCVMoveBackward := FALSE;
									SamesizeCV.M_MoveForward();			
							END_CASE					
				
						END_IF	
				
						IF tonDelay.Q THEN
							tonFeedBoxTimeout.IN :=FALSE;
							uiBothStep:=9000;
						END_IF
						IF tonFeedBoxTimeout.Q THEN
							tonFeedBoxTimeout.IN :=FALSE;
							strStatus :='FB_RobotRegionMove_AllocatedConveyor Step 30000: Feed Box timeout';
							uiResumeStep:=30000;
							_Abort:=TRUE;
						END_IF
				
				9000:
						BoxReady_2nd:=TRUE;
						tonDelay.IN :=FALSE;
						bSameSizeCVMoveForward  :=FALSE;
						bSameSizeCVMoveBackward :=FALSE;
						bDiffCVMoveForward		:=FALSE;
						bDiffCVMoveBackward		:=FALSE;
						DifferenceCV.M_MotorStop();
						SamesizeCV.M_MotorStop();
				
					
       
      	  END_CASE

       	  // Robot Abs move
           		 Robot.M_StartRobotAbsMove( GetBox:=Get,
											UseClampA:=UseA,
											UseClampB:=UseB,
											Area:=Area,
											ClampA_Address:=Address_A,
											ClampB_Address:=Address_B,
											BoxReady_1:=BoxReady_1st,
											BoxReady_2:=BoxReady_2nd);	
		
		
        IF Robot._DI1.Done THEN
			tonTimeOut.IN:=FALSE;
            uiExecutingStep := 30080;
        END_IF
			tonTimeOut.IN:=TRUE;
		IF tonTimeOut.Q=TRUE THEN
			tonTimeOut.IN:=FALSE;
			strStatus :='FB_RobotRegionMove_AllocatedConveyor Step 30000: Robot move timeout';
			_Abort:=TRUE;
		END_IF
		IF Robot._DI1.Error THEN
			_Abort		:= TRUE;
			strStatus	:= CONCAT('FB_RobotRegionMove_AllocatedConveyor Step 30000: ',robot.ErrMsg);
			uiResumeStep:= 30000;
		END_IF
    30080: // Check robot command is clear
        
        Robot.M_ResetRobotAbsMove(UseA,UseB);

        IF NOT Robot._DI1.Done THEN
			tonTimeOut.IN:=FALSE;
            uiExecutingStep := 50000; // go to place step
        END_IF    
   		tonTimeOut.IN:=TRUE;
		IF tonTimeOut.Q=TRUE THEN
			strStatus :='FB_RobotRegionMove_AllocatedConveyor Step 30080: Stop Robot timeout';
			_Error:=TRUE;
		END_IF	
  	50000:	// if robot put need box forward more time
			IF NOT Get THEN
				uiExecutingStep :=51000;
			ELSE
				uiExecutingStep :=99000;
			END_IF
    51000:	//conveyor forward 
			IF UseA THEN
				CASE Address_A OF
					1:
						tonDelay.IN := NOT Input.bDifferentSizeCV_BoxDetect7_Sensor;
						DifferenceCV.M_MoveForward();
					2:
						tonDelay.IN :=NOT SameSizeFullSensor;
						SamesizeCV.M_MoveForward();			
				END_CASE
			END_IF					
			IF UseB THEN
				CASE Address_B OF
					1:
						tonDelay.IN := NOT Input.bDifferentSizeCV_BoxDetect7_Sensor;
						DifferenceCV.M_MoveForward();
					2:
						tonDelay.IN :=NOT SameSizeFullSensor;
						SamesizeCV.M_MoveForward();			
				END_CASE
			END_IF
						IF tonDelay.Q THEN
							tonFeedBoxTimeout.IN :=FALSE;
							uiExecutingStep:=99000;
						END_IF
						IF tonFeedBoxTimeout.Q THEN
							tonFeedBoxTimeout.IN :=FALSE;
							strStatus :='FB_RobotRegionMove_AllocatedConveyor Step 51000: Feed Box timeout';
							uiResumeStep:=30000;
							_Abort:=TRUE;
						END_IF
    99000: // process done
         Status    := 'FB_RobotRegionMove_AllocatedConveyor Step 99000: Process completed';
		 bSameSizeCVMoveForward  :=FALSE;
		 bSameSizeCVMoveBackward :=FALSE;
		 bDiffCVMoveForward		:=FALSE;
		 bDiffCVMoveBackward		:=FALSE;
			 SamesizeCV.M_MotorStop();
			 DifferenceCV.M_MotorStop();
		 cylinder.List.fbSameSizeCV_Press3.M_Retract();
		 cylinder.List.fbSameSizeCV_Press4.M_Retract();
			 
        _Executed := TRUE;
		
END_CASE
IF _Executed THEN
    eState := STATE_DONE;
ELSIF _Error THEN
	eState := STATE_ERROR;
ELSIF NOT Execute THEN
    eState := STATE_RESETTING;
END_IF
IF _Abort OR Abort THEN
	eSTATE:=STATE_ABORTING;
END_IF
END_METHOD

METHOD  M_STATE_RESETTING
VAR_INPUT
END_VAR
// Done := false 更改到Dormant 清除確保，上位檢查到done 後可以直接下Execute

CASE uiResettingStep OF

	0:
		tonTimeOut.IN:=FALSE;
		tonDelay_SameSizeDelayBox.IN :=FALSE;
		TON_CVmovedelay.IN := FALSE;
		Robot.M_ResetAllCommand();
		Robot.M_ResetRobotAbsMove(TRUE,TRUE);
		DifferenceCV.M_MotorStop();
		SamesizeCV.M_MotorStop();
		cylinder.List.fbSameSizeCV_Press3.M_Retract();
		cylinder.List.fbSameSizeCV_Press4.M_Retract();
		uiResettingStep:=100;

	100:

		uiResettingStep:=9999;
	9999:
//		Done := FALSE;
//		Busy := FALSE;
		_ResetCompleted:=TRUE;
END_CASE
IF _ResetCompleted THEN
	eSTATE:=STATE_DORMANT;
END_IF
END_METHOD

END_FUNCTION_BLOCK

// ---- Library/20_MachineUnits/21_StorageArea/Service_Robot/FB_RobotRegionMove_BufferArea.TcPOU
FUNCTION_BLOCK FB_RobotRegionMove_BufferArea EXTENDS FB_ObjectBase_V2 IMPLEMENTS IBasicElement
VAR_INPUT
    Robot : REFERENCE TO FB_FanucRobot_Basic_V2;
    // Command   : ST_WareHouseWithRobotMove_Command;
    Info : ST_RobotRegionMove_Info;
    Stop : BOOL;
END_VAR
VAR_OUTPUT
    // Status : ST_WareHouseWithRobotMove_Status;

END_VAR
VAR
    //_Abort       : BOOL;
    strStatus    : STRING;
    uiResumeStep : UINT;

    Area : E_RobotArea := E_RobotArea.BufferArea;
    UseA : BOOL;
    UseB : BOOL;

    Get               : BOOL;
    tonTimeOut        : TON;
    _UniqueErrorCode  : STRING;
    PreviousStrStatus : STRING;
    PreviousErrorCode : STRING;
	
	_bRetry			  : BOOL;
END_VAR

SUPER^.A10_StateControl();
A00_BasicUnits();

(*============================================================
Create Date : 2026/04/01
Last Update	: 2026/04/01
Change Log  : 2026/04/01，移植泰興鏡射機版本。
============================================================*)

ACTION A00_BasicUnits:
tonTimeOut(PT :=T#60S);
END_ACTION

METHOD M_CheckClampStatus : BOOL
VAR_INPUT
END_VAR
M_CheckClampStatus := FALSE;

IF NOT UseA AND NOT UseB THEN
	M_CheckClampStatus 	:= FALSE;
	strStatus 			:= 'FB_RobotRegionMove_BufferArea: Wrong Command , Both Clammp not used';
	RETURN;
END_IF

IF UseA THEN
	IF Get THEN
		IF NOT Robot._DI1.ClampA_Open THEN
			M_CheckClampStatus  := FALSE;
			strStatus			:= 'FB_RobotRegionMove_BufferArea: Robot Use A Clamp Get ,but Clamp not open ';
			RETURN;
		END_IF
	ELSE
		IF Robot._DI1.ClampA_Open THEN
			M_CheckClampStatus	:= FALSE;
			strStatus			:= 'FB_RobotRegionMove_BufferArea: Robot Use A Clamp Place ,but Clamp open';
			RETURN;
		END_IF
	END_IF
END_IF
IF UseB THEN
	IF Get THEN
		IF NOT Robot._DI1.ClampB_Open THEN
			M_CheckClampStatus  := FALSE;
			strStatus			:= 'FB_RobotRegionMove_BufferArea: Robot Use B Clamp Get ,but Clamp not open ';
			RETURN;
		END_IF
	ELSE
		IF Robot._DI1.ClampB_Open THEN
			M_CheckClampStatus	:= FALSE;
			strStatus			:= 'FB_RobotRegionMove_BufferArea: Robot Use B Clamp Place ,but Clamp open';
			RETURN;
		END_IF
	END_IF
END_IF

M_CheckClampStatus := TRUE;
END_METHOD

METHOD M_CheckCommand : BOOL // True : Command is useful
VAR_INPUT
END_VAR
VAR
	
END_VAR
// Check command paremeter is correct

THIS^.Get :=Info.Get;
UseA := Info.UseA;
UseB := Info.UseB;
//Buffer area
		
IF UseA AND ( Info.A_Position<1 OR  Info.A_Position>40) THEN
	strStatus:='FB_RobotRegionMove_BufferArea: Wrong command ,Position A Not allow';
	M_CheckCommand:=FALSE;
	RETURN;			
END_IF		

IF UseB AND( Info.B_Position<1 OR  Info.B_Position>40 )THEN
	strStatus:='FB_RobotRegionMove_BufferArea: Wrong command ,Position B Not allow';
	M_CheckCommand:=FALSE;
	RETURN;			
END_IF
		
M_CheckCommand:=TRUE;
END_METHOD

METHOD M_CheckUnitsNotBusy : BOOL
VAR_INPUT
END_VAR
M_CheckUnitsNotBusy := true;
END_METHOD

METHOD M_CheckUnitsReady : BOOL
VAR_INPUT
END_VAR
M_CheckUnitsReady := true;
END_METHOD

METHOD  M_STATE_ABORTED
VAR_INPUT
END_VAR
IF NOT _bRetry THEN
	ERROR 	:= TRUE;
	Busy    := FALSE;
	Aborted := TRUE;
	Status 	:= strStatus;
	UniqueErrorCode:= _UniqueErrorCode;
	uiAbortingStep := 0;
	_AbortCompleted:= FALSE;
END_IF
IF reset THEN
	_bRetry := TRUE;
	error   := FALSE;
	Aborted := FALSE;
	_Abort	:= FALSE;
END_IF

IF NOT Execute THEN
	eSTATE:=STATE_RESETTING;
END_IF
IF Execute AND _bRetry AND NOT robot._DI1.Error AND NOT Robot.Halt THEN
	status := '';
	uiExecutingStep :=uiResumeStep;
	PreviousStrStatus := strStatus;
	PreviousErrorCode := _UniqueErrorCode;
	IF GVL_ADS.MachineState <> E_MachineState.Error THEN
		eSTATE:=STATE_EXECUTING;
	END_IF
END_IF
END_METHOD

METHOD  M_STATE_ABORTING
VAR_INPUT
END_VAR
CASE uiAbortingStep OF
	0 :
			tonTimeOut.IN := FALSE;
			_Abort  := FALSE;
			_bRetry	:= FALSE;
			
			IF strStatus = PreviousStrStatus THEN
				_UniqueErrorCode :=PreviousErrorCode;
			END_IF
			uiAbortingStep := 100;
	100:
			IF Robot._DI1.Error THEN
				uiAbortingStep := 200;
			ELSE
				uiAbortingStep := 9999;
			END_IF
	200:		
			 IF DAS_CoreSys.MachineControl.M_RobotResetCmd() THEN
				 uiAbortingStep := 300;
			 END_IF
	300:
			IF DAS_CoreSys.MachineControl.M_RobotStartCmd() THEN
				 uiAbortingStep := 400;
			 END_IF 
	400:
			IF Robot._DI1.Error THEN
		 		uiAbortingStep := 200;
			ELSE
				uiAbortingStep := 9999;
			END_IF
	9999:	
			_AbortCompleted:=TRUE;
END_CASE

IF _AbortCompleted THEN	
	eSTATE :=STATE_ABORTED;
END_IF
END_METHOD

METHOD  M_STATE_DONE
VAR_INPUT
END_VAR
Busy   := FALSE;
_Error := Error := FALSE;
_Abort := Abort := FALSE;
Done   := TRUE;

IF NOT Execute THEN
    eState := STATE_RESETTING;
END_IF
END_METHOD

METHOD  M_STATE_DORMANT
VAR_INPUT
END_VAR
// Clear FB output
Busy            := FALSE;
Done            := FALSE;
Aborted         := FALSE;
Error           := FALSE;
ErrorID         := 0;
Status          := '';
_ResetCompleted := FALSE;
_Error          := FALSE;
_Executed       := FALSE;

tonTimeOut.IN:=FALSE;
strStatus :='No Error';
uiExecutingStep :=uiResettingStep :=uiResumeStep := 0;
uiAbortingStep   := 0;
PreviousStrStatus	:='';
PreviousErrorCode	:='';
_UniqueErrorCode	:='0';
_bRetry				:= false;

// Wait Execute command
IF Execute AND NOT stop THEN
    eState := STATE_EXECUTING;
END_IF
END_METHOD

METHOD  M_STATE_ERROR
VAR_INPUT
END_VAR
ERROR   :=TRUE;
Busy	:=FALSE;
Status := strStatus;
UniqueErrorCode:=_UniqueErrorCode;
IF NOT Execute THEN	
eSTATE:=STATE_RESETTING;
END_IF
END_METHOD

METHOD  M_STATE_EXECUTING
VAR_INPUT
END_VAR
VAR_INST
    ActionMode       : E_ReloadRoundBoxAction;
	BoxReady_1st : BOOL;
	BoxReady_2nd : BOOL;
    CarrierReady_1st : BOOL;
    CarrierReady_2nd : BOOL;
    uiBothStep : UINT;
    uiSingleClampStep : UINT;
	Address_A : INT;
	Address_B : INT;
END_VAR
VAR
	WareHouse: INT;
END_VAR
// Set Busy active edit by johnson
Busy := TRUE;
IF THIS^.Stop THEN // Pending the timeout when Stop signal occur
	tonTimeout.IN :=FALSE;
END_IF
// Service Process
CASE uiExecutingStep OF
	0:
        // Clear variable
        ActionMode       := E_ReloadRoundBoxAction.Undefined;
        CarrierReady_1st := FALSE;
        CarrierReady_2nd := FALSE;
        uiBothStep := 0;
		uiSingleClampStep :=0;
		BoxReady_1st := 0;
		BoxReady_2nd := 0;
		tonTimeOut.IN:=FALSE;
        // Check command
        IF M_CheckCommand() THEN
            uiExecutingStep := 10;
		ELSE
			_Error:=TRUE;
        END_IF
    10:
        // Start process, check units first
        IF M_CheckUnitsReady() THEN
            uiExecutingStep := 20;
        END_IF
    20:
        // CHeck units not busy state
        IF M_CheckUnitsNotBusy() THEN
            uiExecutingStep := 30;
        END_IF

	30:
		IF M_CheckClampStatus() THEN
			uiExecutingStep := 1000;
		ELSE
			_Abort := TRUE;
		END_IF
   
	1000:   
			// Read   coordinate
 			 Address_A := LREAL_TO_INT(Info.A_Position);
			 Address_B := LREAL_TO_INT(Info.B_Position);
			 
			IF UseA AND NOT UseB THEN
				//Only clampA
				uiExecutingStep := 10000;
			ELSIF NOT UseA AND UseB THEN
				//Only ClampB 
				uiExecutingStep := 20000;
			ELSIF UseA AND UseB THEN
				//Both Clamps
				uiExecutingStep := 30000;		
			END_IF
       
    10000: // Only ClampA 
		tonTimeOut.IN:=TRUE;
        IF NOT Robot._DI1.Done THEN            
           		BoxReady_1st:=TRUE;				
			          		 
				  // Robot Abs move
           		 Robot.M_StartRobotAbsMove(GetBox:=Get,
											UseClampA:=UseA,
											UseClampB:=UseB,
											Area:=Area,
											ClampA_Address:=Address_A,
											ClampB_Address:=Address_B,
											BoxReady_1:=BoxReady_1st,
											BoxReady_2:=BoxReady_2nd);	  
		
        ELSE
			tonTimeOut.IN:=FALSE;
            uiExecutingStep := 10080;
        END_IF
			
			IF tonTimeOut.Q=TRUE THEN
				tonTimeOut.IN:=FALSE;			
				uiResumeStep := 10000;			
				strStatus 	 := 'FB_RobotRegionMove_BufferArea Step 10000: Robot Move Timeout';
				_Abort:=TRUE;
			END_IF	
			IF Robot.Error THEN
				tonTimeOut.IN:=FALSE;
				uiResumeStep := 10000;
				strStatus := 'FB_RobotRegionMove_BufferArea Step 10000: ClampA Robot Error';


				_Abort := TRUE;
			END_IF
    10080:
        Robot.M_ResetRobotAbsMove(UseA,UseB); // Clear command and go to place box
		tonTimeOut.IN:=TRUE;
        IF NOT Robot._DI1.Done THEN
			tonTimeOut.IN:=FALSE;
            uiExecutingStep := 99000; 
        END_IF
    	IF tonTimeOut.Q=TRUE THEN
			strStatus :='FB_RobotRegionMove_BufferArea Step 10080: Reset Robot timeout';




			_Error:=TRUE;
		END_IF	
    
   20000: // Only ClampB
			IF NOT Robot._DI1.Done THEN           		
					BoxReady_2nd:=TRUE;				          		 
					  // Robot Abs move
					 Robot.M_StartRobotAbsMove( GetBox:=Get,
												UseClampA:=UseA,
												UseClampB:=UseB,
												Area:=Area,
												ClampA_Address:=Address_A,
												ClampB_Address:=Address_B,
												BoxReady_1:=BoxReady_1st,
												BoxReady_2:=BoxReady_2nd);	
			ELSE
				tonTimeOut.IN:=FALSE;
				uiExecutingStep := 20080;
			END_IF
				tonTimeOut.IN:=TRUE;
			IF tonTimeOut.Q=TRUE THEN
				tonTimeOut.IN:=FALSE;			
				uiResumeStep := 20000;		
				strStatus := 'FB_RobotRegionMove_BufferArea Step 20000: Robot Move Timeout';
				_Abort:=TRUE;
			END_IF	
			IF Robot.Error THEN
				tonTimeOut.IN:=FALSE;
				uiResumeStep := 20000;
				strStatus := 'FB_RobotRegionMove_BufferArea Step 20000: Use ClampB Robot Error';


				_Abort := TRUE;
			END_IF
    20080:
			   Robot.M_ResetRobotAbsMove(UseA,UseB);; // Clear command 
		
				IF NOT Robot._DI1.Done THEN
					uiExecutingStep := 99000; 
				END_IF
				tonTimeOut.IN:=TRUE;
				IF tonTimeOut.Q=TRUE THEN
					strStatus :='FB_RobotRegionMove_BufferArea Step 20080: Reset Robot timeout';




					_Error:=TRUE;
				END_IF	
    30000: // Both Clamps
        		
		
		  CASE uiBothStep OF
           		0://	
					BoxReady_1st := FALSE;
					BoxReady_2nd := FALSE;					
					uiBothStep:=1000;	
	
				1000:
						BoxReady_1st:=TRUE;
						uiBothStep:=2000;
						
				2000:
						IF Robot._DI1.Notification THEN
							uiBothStep:=3000;
						END_IF
				3000:
					
					
						uiBothStep:=9000;	
					
				9000:
						BoxReady_2nd:=TRUE;
						uiBothStep:=9999;
				
				9999: //Wait		
        // wait reset
        END_CASE

       	  // Robot Abs move
           		 Robot.M_StartRobotAbsMove( GetBox:=Get,
											UseClampA:=UseA,
											UseClampB:=UseB,
											Area:=Area,
											ClampA_Address:=Address_A,
											ClampB_Address:=Address_B,
											BoxReady_1:=BoxReady_1st,
											BoxReady_2:=BoxReady_2nd);	
		
		
        IF Robot._DI1.Done THEN
			tonTimeOut.IN:=FALSE;
            uiExecutingStep := 30080;
        END_IF
		IF tonTimeOut.Q  THEN
			tonTimeOut.IN:=FALSE;			
			strStatus := 'FB_RobotRegionMove_BufferArea Step 30000: Robot Move Timeout';
			uiResumeStep     := 30000;
			_Abort:=TRUE;
		END_IF	
		IF Robot.Error THEN
			uiResumeStep     := 30000;
			_Abort := TRUE;
			strStatus :='FB_RobotRegionMove_BufferArea Step 30000: Use bothClamp robot Error';


		END_IF
		
		
    30080: // Check robot command is clear
        
        Robot.M_ResetRobotAbsMove(UseA,UseB);

        IF NOT Robot._DI1.Done THEN
			tonTimeOut.IN:=FALSE;
            uiExecutingStep := 99000; // go to place step
        END_IF    
   		tonTimeOut.IN:=TRUE;
		IF tonTimeOut.Q=TRUE THEN
			strStatus :='FB_RobotRegionMove_BufferArea Step 30080: Stop Robot timeout';
			_Error:=TRUE;
		END_IF	
   
    99000: // process done
                Status    := 'FB_RobotRegionMove_BufferArea Step 99000: Process completed';
        _Executed := TRUE;
END_CASE

IF _Executed THEN
    eState := STATE_DONE;
ELSIF _Error THEN

    eState := STATE_ERROR;
ELSIF NOT Execute THEN
    eState := STATE_RESETTING;
END_IF
IF _Abort OR Abort THEN

	eSTATE:=STATE_ABORTING;
END_IF
END_METHOD

METHOD  M_STATE_RESETTING
VAR_INPUT
END_VAR
// Done := false 更改到Dormant 清除確保，上位檢查到done 後可以直接下Execute

CASE uiResettingStep OF

	0:
		tonTimeOut.IN:=FALSE;
		Robot.M_ResetAllCommand();
		Robot.M_ResetRobotAbsMove(TRUE,TRUE);

		uiResettingStep:=9999;
	9999:
//		Done := FALSE;
//		Busy := FALSE;
		_ResetCompleted:=TRUE;
END_CASE
IF _ResetCompleted THEN
	eSTATE:=STATE_DORMANT;
END_IF
END_METHOD

END_FUNCTION_BLOCK

// ---- Library/20_MachineUnits/21_StorageArea/Service_Robot/FB_RobotRegionMove_RoundBelt.TcPOU
FUNCTION_BLOCK FB_RobotRegionMove_RoundBelt EXTENDS FB_ObjectBase_V2 IMPLEMENTS IBasicElement
VAR_INPUT
    Robot     					: REFERENCE TO FB_FanucRobot_Basic_V2;
	RoundBelt					: REFERENCE TO FB_RoundBeltService;	
   // Command   : ST_WareHouseWithRobotMove_Command;
    Info	  : ST_RobotRegionMove_Info;
	Input : ST_InputTable;
	Stop	  : BOOL;
END_VAR
VAR_OUTPUT
  // Status : ST_WareHouseWithRobotMove_Status;
END_VAR
VAR
	//_Abort		: BOOL;
	strStatus	: STRING;
	uiResumeStep : UINT;
	
	Area	: E_RobotArea :=E_RobotArea.RoundBelt;
	UseA 	: BOOL;
	UseB	: BOOL;
	
	Get 	:BOOL;
	tonTimeOut	:TON;
	tonCheckRoundBeltDelay	:TON;
	_UniqueErrorCode :STRING;
	PreviousStrStatus : STRING;
	PreviousErrorCode : STRING;
	
	_bRetry	: BOOL;
END_VAR

SUPER^.A10_StateControl();
A00_BasicUnits();

ACTION A00_BasicUnits:
tonTimeOut(PT:=T#60S);
tonCheckRoundBeltDelay(PT:=T#2S);
ErrorID:=2220;
END_ACTION

METHOD M_CheckClampStatus : BOOL
VAR_INPUT
END_VAR
M_CheckClampStatus := FALSE;

IF NOT UseA AND NOT UseB THEN
	M_CheckClampStatus 	:= FALSE;
	strStatus 			:= 'FB_RobotRegionMove_RoundBelt: Wrong Command , Both Clammp not used';
	RETURN;
END_IF

IF UseA THEN
	IF Get THEN
		IF NOT Robot._DI1.ClampA_Open THEN
			M_CheckClampStatus  := FALSE;
			strStatus			:= 'FB_RobotRegionMove_RoundBelt: Robot Use A Clamp Get ,but Clamp not open ';
			RETURN;
		END_IF
	ELSE
		IF Robot._DI1.ClampA_Open THEN
			M_CheckClampStatus	:= FALSE;
			strStatus			:= 'FB_RobotRegionMove_RoundBelt: Robot Use A Clamp Place ,but Clamp open';
			RETURN;
		END_IF
	END_IF
END_IF
IF UseB THEN
	IF Get THEN
		IF NOT Robot._DI1.ClampB_Open THEN
			M_CheckClampStatus  := FALSE;
			strStatus			:= 'FB_RobotRegionMove_RoundBelt: Robot Use B Clamp Get ,but Clamp not open ';
			RETURN;
		END_IF
	ELSE
		IF Robot._DI1.ClampB_Open THEN
			M_CheckClampStatus	:= FALSE;
			strStatus			:= 'FB_RobotRegionMove_RoundBelt: Robot Use B Clamp Place ,but Clamp open';
			RETURN;
		END_IF
	END_IF
END_IF

M_CheckClampStatus := TRUE;
END_METHOD

METHOD M_CheckCommand : BOOL // True : Command is useful
VAR_INPUT
END_VAR
VAR
	
END_VAR
// Check command paremeter is correct
	
THIS^.Get :=Info.Get;
UseA := Info.UseA;
UseB := Info.UseB;
	//Normal command : RoundBelt
		IF Info.UseA AND (Info.A_Position<1 OR  Info.A_Position>3) THEN
			strStatus:='FB_RobotRegionMove_RoundBelt: Wrong command ,Position A Not allowed';
			M_CheckCommand:=FALSE;
			RETURN;			
		END_IF
		
	
	//Normal command : RoundBelt
		IF Info.UseB AND(Info.B_Position<1 OR  Info.B_Position>3) THEN
			strStatus:='FB_RobotRegionMove_RoundBelt: Wrong command ,Position B Not allowed';
			M_CheckCommand:=FALSE;
			RETURN;				
		END_IF
		
	

M_CheckCommand:=TRUE;
END_METHOD

METHOD M_CheckUnitsNotBusy : BOOL
VAR_INPUT
END_VAR
M_CheckUnitsNotBusy := true;
END_METHOD

METHOD M_CheckUnitsReady : BOOL
VAR_INPUT
END_VAR
M_CheckUnitsReady := true;
END_METHOD

METHOD  M_STATE_ABORTED
VAR_INPUT
END_VAR
IF NOT _bRetry THEN
	ERROR 	:= TRUE;
	Busy    := FALSE;
	Aborted := TRUE;
	Status 	:= strStatus;
	UniqueErrorCode := _UniqueErrorCode;
	uiAbortingStep 		:= 0;
	_AbortCompleted		:= FALSE;
END_IF

